LIN {X 0,Y 408.559,Z 372.352,A -85,B 0,C 180,E1 18045.699,E2 18045.699} C_VEL
LIN {X 0,Y 407.046,Z 362.331,A -85,B 0,C 180,E1 18045.227,E2 18045.227} C_VEL
LIN {X 0,Y 396.72,Z 344.882,A -85,B 0,C 180,E1 18043.129,E2 18043.129} C_VEL
LIN {X 0,Y 386.297,Z 328.726,A -85,B 0,C 180,E1 18040.835,E2 18040.835} C_VEL
LIN {X 0,Y 381.778,Z 321.934,A -85,B 0,C 180,E1 18039.72,E2 18039.72} C_VEL
LIN {X 0,Y 376.078,Z 309.997,A -85,B 0,C 180,E1 18036.741,E2 18036.741} C_VEL
LIN {X 0,Y 371.702,Z 301.451,A -85,B 0,C 180,E1 18034.331,E2 18034.331} C_VEL
LIN {X 0,Y 369.056,Z 296.536,A -85,B 0,C 180,E1 18032.81,E2 18032.81} C_VEL
LIN {X 0,Y 366.734,Z 292.115,A -85,B 0,C 180,E1 18031.382,E2 18031.382} C_VEL
LIN {X 0,Y 364.759,Z 288.388,A -85,B 0,C 180,E1 18030.108,E2 18030.108} C_VEL
LIN {X 0,Y 362.046,Z 283.882,A -85,B 0,C 180,E1 18028.36,E2 18028.36} C_VEL
LIN {X 0,Y 361.832,Z 282.774,A -85,B 0,C 180,E1 18027.84,E2 18027.84} C_VEL
LIN {X 0,Y 361.811,Z 282.657,A -85,B 0,C 180,E1 18023.623,E2 18023.623} C_VEL
LIN {X 0,Y 361.809,Z 282.653,A -85,B 0,C 180,E1 18019.535,E2 18019.535} C_VEL
LIN {X 0,Y 361.808,Z 282.65,A -85,B 0,C 180,E1 18015.327,E2 18015.327} C_VEL
LIN {X 0,Y 361.791,Z 282.651,A -85,B 0,C 180,E1 18011.155,E2 18011.155} C_VEL
LIN {X 0,Y 361.78,Z 282.655,A -85,B 0,C 180,E1 18006.985,E2 18006.985} C_VEL
LIN {X 0,Y 361.77,Z 282.662,A -85,B 0,C 180,E1 18002.852,E2 18002.852} C_VEL
LIN {X 0,Y 361.762,Z 282.669,A -85,B 0,C 180,E1 17998.733,E2 17998.733} C_VEL
LIN {X 0,Y 361.753,Z 282.674,A -85,B 0,C 180,E1 17994.608,E2 17994.608} C_VEL
LIN {X 0,Y 361.748,Z 282.675,A -85,B 0,C 180,E1 17990.615,E2 17990.615} C_VEL
LIN {X 0,Y 361.742,Z 282.675,A -85,B 0,C 180,E1 17986.575,E2 17986.575} C_VEL
LIN {X 0,Y 361.74,Z 282.674,A -85,B 0,C 180,E1 17982.466,E2 17982.466} C_VEL
LIN {X 0,Y 361.746,Z 282.671,A -85,B 0,C 180,E1 17978.432,E2 17978.432} C_VEL
LIN {X 0,Y 361.819,Z 282.907,A -85,B 0,C 180,E1 17975.163,E2 17975.163} C_VEL
LIN {X 0,Y 363.332,Z 286.523,A -85,B 0,C 180,E1 17973.877,E2 17973.877} C_VEL
LIN {X 0,Y 364.801,Z 288.276,A -85,B 0,C 180,E1 17973.113,E2 17973.113} C_VEL
LIN {X 0,Y 366.755,Z 292.174,A -85,B 0,C 180,E1 17971.86,E2 17971.86} C_VEL
LIN {X 0,Y 367.885,Z 293.939,A -85,B 0,C 180,E1 17971.246,E2 17971.246} C_VEL
LIN {X 0,Y 370.686,Z 299.01,A -85,B 0,C 180,E1 17969.668,E2 17969.668} C_VEL
LIN {X 0,Y 375.284,Z 307.456,A -85,B 0,C 180,E1 17967.259,E2 17967.259} C_VEL
LIN {X 0,Y 376.894,Z 310.291,A -85,B 0,C 180,E1 17966.646,E2 17966.646} C_VEL
LIN {X 0,Y 385.998,Z 322.591,A -85,B 0,C 180,E1 17964.442,E2 17964.442} C_VEL
LIN {X 0,Y 396.684,Z 338.125,A -85,B 0,C 180,E1 17962.073,E2 17962.073} C_VEL
LIN {X 0,Y 408.24,Z 356.697,A -85,B 0,C 180,E1 17959.716,E2 17959.716} C_VEL
LIN {X 0,Y 411.508,Z 362.693,A -85,B 0,C 180,E1 17959.072,E2 17959.072} C_VEL
LIN {X 0,Y 402.389,Z 573.786,A -85,B 0,C 180,E1 17954.935,E2 17954.935} C_VEL
LIN {X 0,Y 400.703,Z 607.918,A -85,B 0,C 180,E1 17954.213,E2 17954.213} C_VEL
LIN {X 0,Y 398.591,Z 630.344,A -85,B 0,C 180,E1 17953.522,E2 17953.522} C_VEL
LIN {X 0,Y 395.913,Z 651.73,A -85,B 0,C 180,E1 17952.594,E2 17952.594} C_VEL
LIN {X 0,Y 392.818,Z 672.423,A -85,B 0,C 180,E1 17951.435,E2 17951.435} C_VEL
LIN {X 0,Y 389.456,Z 691.906,A -85,B 0,C 180,E1 17950.088,E2 17950.088} C_VEL
LIN {X 0,Y 385.56,Z 711.788,A -85,B 0,C 180,E1 17948.394,E2 17948.394} C_VEL
LIN {X 0,Y 381.679,Z 730.327,A -85,B 0,C 180,E1 17946.487,E2 17946.487} C_VEL
LIN {X 0,Y 377.741,Z 748.111,A -85,B 0,C 180,E1 17944.318,E2 17944.318} C_VEL
LIN {X 0,Y 373.949,Z 765.002,A -85,B 0,C 180,E1 17941.874,E2 17941.874} C_VEL
LIN {X 0,Y 370.47,Z 780.284,A -85,B 0,C 180,E1 17939.241,E2 17939.241} C_VEL
LIN {X 0,Y 367.358,Z 794.572,A -85,B 0,C 180,E1 17936.336,E2 17936.336} C_VEL
LIN {X 0,Y 364.783,Z 807.38,A -85,B 0,C 180,E1 17933.246,E2 17933.246} C_VEL
LIN {X 0,Y 362.879,Z 818.173,A -85,B 0,C 180,E1 17930.146,E2 17930.146} C_VEL
LIN {X 0,Y 361.483,Z 827.462,A -85,B 0,C 180,E1 17926.883,E2 17926.883} C_VEL
LIN {X 0,Y 360.594,Z 835.304,A -85,B 0,C 180,E1 17923.468,E2 17923.468} C_VEL
LIN {X 0,Y 360.17,Z 841.103,A -85,B 0,C 180,E1 17920.234,E2 17920.234} C_VEL
LIN {X 0,Y 360.026,Z 845.162,A -85,B 0,C 180,E1 17917.019,E2 17917.019} C_VEL
LIN {X 0,Y 359.994,Z 847.849,A -85,B 0,C 180,E1 17913.662,E2 17913.662} C_VEL
LIN {X 0,Y 360.004,Z 848.78,A -85,B 0,C 180,E1 17910.796,E2 17910.796} C_VEL
LIN {X 0,Y 359.999,Z 848.431,A -85,B 0,C 180,E1 17907.612,E2 17907.612} C_VEL
LIN {X 0,Y 360.003,Z 846.641,A -85,B 0,C 180,E1 17904.582,E2 17904.582} C_VEL
LIN {X 0,Y 360.072,Z 843.093,A -85,B 0,C 180,E1 17901.215,E2 17901.215} C_VEL
LIN {X 0,Y 360.343,Z 838.399,A -85,B 0,C 180,E1 17898.151,E2 17898.151} C_VEL
LIN {X 0,Y 360.95,Z 831.803,A -85,B 0,C 180,E1 17894.907,E2 17894.907} C_VEL
LIN {X 0,Y 362.036,Z 823.526,A -85,B 0,C 180,E1 17891.649,E2 17891.649} C_VEL
LIN {X 0,Y 363.704,Z 813.284,A -85,B 0,C 180,E1 17888.385,E2 17888.385} C_VEL
LIN {X 0,Y 365.916,Z 801.567,A -85,B 0,C 180,E1 17885.288,E2 17885.288} C_VEL
LIN {X 0,Y 368.825,Z 787.697,A -85,B 0,C 180,E1 17882.208,E2 17882.208} C_VEL
LIN {X 0,Y 372.076,Z 773.156,A -85,B 0,C 180,E1 17879.478,E2 17879.478} C_VEL
LIN {X 0,Y 375.715,Z 757.109,A -85,B 0,C 180,E1 17876.939,E2 17876.939} C_VEL
LIN {X 0,Y 379.502,Z 740.143,A -85,B 0,C 180,E1 17874.67,E2 17874.67} C_VEL
LIN {X 0,Y 383.602,Z 721.198,A -85,B 0,C 180,E1 17872.537,E2 17872.537} C_VEL
LIN {X 0,Y 387.425,Z 702.563,A -85,B 0,C 180,E1 17870.782,E2 17870.782} C_VEL
LIN {X 0,Y 390.927,Z 683.359,A -85,B 0,C 180,E1 17869.293,E2 17869.293} C_VEL
LIN {X 0,Y 394.328,Z 662.52,A -85,B 0,C 180,E1 17867.981,E2 17867.981} C_VEL
LIN {X 0,Y 397.271,Z 641.356,A -85,B 0,C 180,E1 17866.929,E2 17866.929} C_VEL
LIN {X 0,Y 399.587,Z 620.581,A -85,B 0,C 180,E1 17866.155,E2 17866.155} C_VEL
LIN {X 0,Y 401.273,Z 598.399,A -85,B 0,C 180,E1 17865.57,E2 17865.57} C_VEL
LIN {X 0,Y 410.569,Z 383.446,A -85,B 0,C 180,E1 17861.338,E2 17861.338} C_VEL
LIN {X 0,Y 411.329,Z 362.088,A -85,B 0,C 180,E1 17860.897,E2 17860.897} C_VEL
LIN {X 0,Y 401.183,Z 345.219,A -85,B 0,C 180,E1 17858.883,E2 17858.883} C_VEL
LIN {X 0,Y 390.845,Z 329.535,A -85,B 0,C 180,E1 17856.679,E2 17856.679} C_VEL
LIN {X 0,Y 381.262,Z 316.025,A -85,B 0,C 180,E1 17854.458,E2 17854.458} C_VEL
LIN {X 0,Y 375.815,Z 308.655,A -85,B 0,C 180,E1 17853.052,E2 17853.052} C_VEL
LIN {X 0,Y 372.269,Z 301.954,A -85,B 0,C 180,E1 17851.223,E2 17851.223} C_VEL
LIN {X 0,Y 369.727,Z 297.293,A -85,B 0,C 180,E1 17849.841,E2 17849.841} C_VEL
LIN {X 0,Y 366.999,Z 292.443,A -85,B 0,C 180,E1 17848.297,E2 17848.297} C_VEL
LIN {X 0,Y 364.933,Z 288.721,A -85,B 0,C 180,E1 17847.053,E2 17847.053} C_VEL
LIN {X 0,Y 363.842,Z 287.108,A -85,B 0,C 180,E1 17846.435,E2 17846.435} C_VEL
LIN {X 0,Y 362.104,Z 284.18,A -85,B 0,C 180,E1 17845.34,E2 17845.34} C_VEL
LIN {X 0,Y 361.813,Z 282.858,A -85,B 0,C 180,E1 17844.837,E2 17844.837} C_VEL
LIN {X 0,Y 361.785,Z 282.663,A -85,B 0,C 180,E1 17840.886,E2 17840.886} C_VEL
LIN {X 0,Y 361.775,Z 282.657,A -85,B 0,C 180,E1 17836.704,E2 17836.704} C_VEL
LIN {X 0,Y 361.771,Z 282.657,A -85,B 0,C 180,E1 17832.611,E2 17832.611} C_VEL
LIN {X 0,Y 361.769,Z 282.659,A -85,B 0,C 180,E1 17828.423,E2 17828.423} C_VEL
LIN {X 0,Y 361.776,Z 282.665,A -85,B 0,C 180,E1 17824.438,E2 17824.438} C_VEL
LIN {X 0,Y 361.777,Z 282.669,A -85,B 0,C 180,E1 17820.316,E2 17820.316} C_VEL
LIN {X 0,Y 361.777,Z 282.672,A -85,B 0,C 180,E1 17816.196,E2 17816.196} C_VEL
LIN {X 0,Y 361.778,Z 282.672,A -85,B 0,C 180,E1 17812.057,E2 17812.057} C_VEL
LIN {X 0,Y 361.774,Z 282.671,A -85,B 0,C 180,E1 17807.875,E2 17807.875} C_VEL
LIN {X 0,Y 361.779,Z 282.668,A -85,B 0,C 180,E1 17803.791,E2 17803.791} C_VEL
LIN {X 0,Y 361.781,Z 282.67,A -85,B 0,C 180,E1 17799.621,E2 17799.621} C_VEL
LIN {X 0,Y 361.784,Z 282.669,A -85,B 0,C 180,E1 17795.399,E2 17795.399} C_VEL
LIN {X 0,Y 361.829,Z 282.875,A -85,B 0,C 180,E1 17791.875,E2 17791.875} C_VEL
LIN {X 0,Y 363.175,Z 286.201,A -85,B 0,C 180,E1 17790.656,E2 17790.656} C_VEL
LIN {X 0,Y 364.832,Z 288.623,A -85,B 0,C 180,E1 17789.685,E2 17789.685} C_VEL
LIN {X 0,Y 366.815,Z 292.212,A -85,B 0,C 180,E1 17788.442,E2 17788.442} C_VEL
LIN {X 0,Y 370.235,Z 298.661,A -85,B 0,C 180,E1 17786.384,E2 17786.384} C_VEL
LIN {X 0,Y 374.748,Z 307.279,A -85,B 0,C 180,E1 17783.868,E2 17783.868} C_VEL
LIN {X 0,Y 380.66,Z 319.547,A -85,B 0,C 180,E1 17780.726,E2 17780.726} C_VEL
LIN {X 0,Y 382.582,Z 323.315,A -85,B 0,C 180,E1 17779.917,E2 17779.917} C_VEL
LIN {X 0,Y 394.621,Z 341.47,A -85,B 0,C 180,E1 17777.206,E2 17777.206} C_VEL
LIN {X 0,Y 405.534,Z 359.797,A -85,B 0,C 180,E1 17774.959,E2 17774.959} C_VEL
LIN {X 0,Y 407.24,Z 363.206,A -85,B 0,C 180,E1 17774.613,E2 17774.613} C_VEL
LIN {X 0,Y 408.507,Z 373.825,A -85,B 0,C 180,E1 17774.166,E2 17774.166} C_VEL
LIN {X 0,Y 400.581,Z 595.446,A -85,B 0,C 180,E1 17770.128,E2 17770.128} C_VEL
LIN {X 0,Y 398.92,Z 616.173,A -85,B 0,C 180,E1 17769.518,E2 17769.518} C_VEL
LIN {X 0,Y 396.654,Z 635.991,A -85,B 0,C 180,E1 17768.691,E2 17768.691} C_VEL
LIN {X 0,Y 393.787,Z 655.659,A -85,B 0,C 180,E1 17767.608,E2 17767.608} C_VEL
LIN {X 0,Y 390.647,Z 673.719,A -85,B 0,C 180,E1 17766.354,E2 17766.354} C_VEL
LIN {X 0,Y 387.043,Z 691.567,A -85,B 0,C 180,E1 17764.813,E2 17764.813} C_VEL
LIN {X 0,Y 383.227,Z 708.408,A -85,B 0,C 180,E1 17763.044,E2 17763.044} C_VEL
LIN {X 0,Y 379.18,Z 724.954,A -85,B 0,C 180,E1 17760.943,E2 17760.943} C_VEL
LIN {X 0,Y 375.312,Z 739.918,A -85,B 0,C 180,E1 17758.654,E2 17758.654} C_VEL
LIN {X 0,Y 371.752,Z 753.448,A -85,B 0,C 180,E1 17756.173,E2 17756.173} C_VEL
LIN {X 0,Y 368.381,Z 766.177,A -85,B 0,C 180,E1 17753.345,E2 17753.345} C_VEL
LIN {X 0,Y 365.69,Z 776.731,A -85,B 0,C 180,E1 17750.485,E2 17750.485} C_VEL
LIN {X 0,Y 363.471,Z 786.215,A -85,B 0,C 180,E1 17747.34,E2 17747.34} C_VEL
LIN {X 0,Y 361.885,Z 794.048,A -85,B 0,C 180,E1 17744.071,E2 17744.071} C_VEL
LIN {X 0,Y 361.143,Z 798.41,A -85,B 0,C 180,E1 17741.796,E2 17741.796} C_VEL
LIN {X 0,Y 359.88,Z 800.467,A -85,B 0,C 180,E1 17740.624,E2 17740.624} C_VEL
LIN {X 0,Y 353.022,Z 805.15,A -85,B 0,C 180,E1 17737.373,E2 17737.373} C_VEL
LIN {X 0,Y 352.29,Z 806.085,A -85,B 0,C 180,E1 17736.396,E2 17736.396} C_VEL
LIN {X 0,Y 352.114,Z 808.279,A -85,B 0,C 180,E1 17732.93,E2 17732.93} C_VEL
LIN {X 0,Y 352.084,Z 808.901,A -85,B 0,C 180,E1 17729.675,E2 17729.675} C_VEL
LIN {X 0,Y 352.129,Z 808.066,A -85,B 0,C 180,E1 17726.419,E2 17726.419} C_VEL
LIN {X 0,Y 352.319,Z 805.768,A -85,B 0,C 180,E1 17723.155,E2 17723.155} C_VEL
LIN {X 0,Y 352.805,Z 801.779,A -85,B 0,C 180,E1 17719.715,E2 17719.715} C_VEL
LIN {X 0,Y 353.7,Z 796.383,A -85,B 0,C 180,E1 17716.431,E2 17716.431} C_VEL
LIN {X 0,Y 355.283,Z 788.833,A -85,B 0,C 180,E1 17712.982,E2 17712.982} C_VEL
LIN {X 0,Y 357.501,Z 779.638,A -85,B 0,C 180,E1 17709.709,E2 17709.709} C_VEL
LIN {X 0,Y 360.209,Z 769.371,A -85,B 0,C 180,E1 17706.749,E2 17706.749} C_VEL
LIN {X 0,Y 363.542,Z 757.357,A -85,B 0,C 180,E1 17703.894,E2 17703.894} C_VEL
LIN {X 0,Y 367.143,Z 744.548,A -85,B 0,C 180,E1 17701.361,E2 17701.361} C_VEL
LIN {X 0,Y 371.241,Z 729.73,A -85,B 0,C 180,E1 17698.922,E2 17698.922} C_VEL
LIN {X 0,Y 375.443,Z 713.556,A -85,B 0,C 180,E1 17696.73,E2 17696.73} C_VEL
LIN {X 0,Y 379.489,Z 696.764,A -85,B 0,C 180,E1 17694.853,E2 17694.853} C_VEL
LIN {X 0,Y 383.437,Z 678.576,A -85,B 0,C 180,E1 17693.182,E2 17693.182} C_VEL
LIN {X 0,Y 386.84,Z 660.766,A -85,B 0,C 180,E1 17691.85,E2 17691.85} C_VEL
LIN {X 0,Y 389.931,Z 641.542,A -85,B 0,C 180,E1 17690.703,E2 17690.703} C_VEL
LIN {X 0,Y 392.484,Z 621.377,A -85,B 0,C 180,E1 17689.796,E2 17689.796} C_VEL
LIN {X 0,Y 394.345,Z 600.962,A -85,B 0,C 180,E1 17689.134,E2 17689.134} C_VEL
LIN {X 0,Y 395.679,Z 573.766,A -85,B 0,C 180,E1 17688.565,E2 17688.565} C_VEL
LIN {X 0,Y 403.042,Z 373.798,A -85,B 0,C 180,E1 17684.893,E2 17684.893} C_VEL
LIN {X 0,Y 401.891,Z 366.492,A -85,B 0,C 180,E1 17684.53,E2 17684.53} C_VEL
LIN {X 0,Y 392.227,Z 349.993,A -85,B 0,C 180,E1 17682.496,E2 17682.496} C_VEL
LIN {X 0,Y 382.017,Z 333.999,A -85,B 0,C 180,E1 17680.169,E2 17680.169} C_VEL
LIN {X 0,Y 373.505,Z 321.545,A -85,B 0,C 180,E1 17678.003,E2 17678.003} C_VEL
LIN {X 0,Y 368.505,Z 311.291,A -85,B 0,C 180,E1 17675.247,E2 17675.247} C_VEL
LIN {X 0,Y 364.257,Z 302.957,A -85,B 0,C 180,E1 17672.735,E2 17672.735} C_VEL
LIN {X 0,Y 361.662,Z 298.135,A -85,B 0,C 180,E1 17671.131,E2 17671.131} C_VEL
LIN {X 0,Y 359.22,Z 293.573,A -85,B 0,C 180,E1 17669.516,E2 17669.516} C_VEL
LIN {X 0,Y 357.062,Z 289.858,A -85,B 0,C 180,E1 17668.063,E2 17668.063} C_VEL
LIN {X 0,Y 356.124,Z 288.304,A -85,B 0,C 180,E1 17667.416,E2 17667.416} C_VEL
LIN {X 0,Y 354.132,Z 284.926,A -85,B 0,C 180,E1 17665.953,E2 17665.953} C_VEL
LIN {X 0,Y 353.888,Z 283.8,A -85,B 0,C 180,E1 17665.433,E2 17665.433} C_VEL
LIN {X 0,Y 353.87,Z 283.643,A -85,B 0,C 180,E1 17661.376,E2 17661.376} C_VEL
LIN {X 0,Y 353.862,Z 283.647,A -85,B 0,C 180,E1 17657.251,E2 17657.251} C_VEL
LIN {X 0,Y 353.851,Z 283.648,A -85,B 0,C 180,E1 17653.065,E2 17653.065} C_VEL
LIN {X 0,Y 353.84,Z 283.646,A -85,B 0,C 180,E1 17648.941,E2 17648.941} C_VEL
LIN {X 0,Y 353.832,Z 283.643,A -85,B 0,C 180,E1 17644.863,E2 17644.863} C_VEL
LIN {X 0,Y 353.826,Z 283.64,A -85,B 0,C 180,E1 17640.81,E2 17640.81} C_VEL
LIN {X 0,Y 353.82,Z 283.639,A -85,B 0,C 180,E1 17636.76,E2 17636.76} C_VEL
LIN {X 0,Y 353.813,Z 283.639,A -85,B 0,C 180,E1 17632.694,E2 17632.694} C_VEL
LIN {X 0,Y 353.804,Z 283.64,A -85,B 0,C 180,E1 17628.591,E2 17628.591} C_VEL
LIN {X 0,Y 353.794,Z 283.641,A -85,B 0,C 180,E1 17624.426,E2 17624.426} C_VEL
LIN {X 0,Y 353.799,Z 283.643,A -85,B 0,C 180,E1 17620.177,E2 17620.177} C_VEL
LIN {X 0,Y 353.876,Z 284.009,A -85,B 0,C 180,E1 17617.578,E2 17617.578} C_VEL
LIN {X 0,Y 355.542,Z 287.711,A -85,B 0,C 180,E1 17616.112,E2 17616.112} C_VEL
LIN {X 0,Y 356.945,Z 289.23,A -85,B 0,C 180,E1 17615.332,E2 17615.332} C_VEL
LIN {X 0,Y 358.676,Z 292.941,A -85,B 0,C 180,E1 17614.046,E2 17614.046} C_VEL
LIN {X 0,Y 360.054,Z 294.855,A -85,B 0,C 180,E1 17613.265,E2 17613.265} C_VEL
LIN {X 0,Y 362.059,Z 298.589,A -85,B 0,C 180,E1 17612,E2 17612} C_VEL
LIN {X 0,Y 363.339,Z 301.047,A -85,B 0,C 180,E1 17611.212,E2 17611.212} C_VEL
LIN {X 0,Y 365.828,Z 305.453,A -85,B 0,C 180,E1 17609.808,E2 17609.808} C_VEL
LIN {X 0,Y 368.266,Z 309.707,A -85,B 0,C 180,E1 17608.582,E2 17608.582} C_VEL
LIN {X 0,Y 379.261,Z 324.47,A -85,B 0,C 180,E1 17605.701,E2 17605.701} C_VEL
LIN {X 0,Y 389.526,Z 339.289,A -85,B 0,C 180,E1 17603.291,E2 17603.291} C_VEL
LIN {X 0,Y 400.953,Z 357.285,A -85,B 0,C 180,E1 17600.837,E2 17600.837} C_VEL
LIN {X 0,Y 405.886,Z 366.065,A -85,B 0,C 180,E1 17599.828,E2 17599.828} C_VEL
LIN {X 0,Y 396.319,Z 578.508,A -85,B 0,C 180,E1 17595.625,E2 17595.625} C_VEL
LIN {X 0,Y 394.662,Z 609.067,A -85,B 0,C 180,E1 17594.957,E2 17594.957} C_VEL
LIN {X 0,Y 392.467,Z 631.269,A -85,B 0,C 180,E1 17594.256,E2 17594.256} C_VEL
LIN {X 0,Y 389.727,Z 652.133,A -85,B 0,C 180,E1 17593.335,E2 17593.335} C_VEL
LIN {X 0,Y 386.508,Z 672.676,A -85,B 0,C 180,E1 17592.166,E2 17592.166} C_VEL
LIN {X 0,Y 382.961,Z 692.287,A -85,B 0,C 180,E1 17590.787,E2 17590.787} C_VEL
LIN {X 0,Y 378.949,Z 711.885,A -85,B 0,C 180,E1 17589.093,E2 17589.093} C_VEL
LIN {X 0,Y 374.886,Z 730.347,A -85,B 0,C 180,E1 17587.163,E2 17587.163} C_VEL
LIN {X 0,Y 370.623,Z 748.64,A -85,B 0,C 180,E1 17584.884,E2 17584.884} C_VEL
LIN {X 0,Y 366.771,Z 764.903,A -85,B 0,C 180,E1 17582.482,E2 17582.482} C_VEL
LIN {X 0,Y 363.011,Z 780.59,A -85,B 0,C 180,E1 17579.72,E2 17579.72} C_VEL
LIN {X 0,Y 359.875,Z 794.16,A -85,B 0,C 180,E1 17576.894,E2 17576.894} C_VEL
LIN {X 0,Y 357.157,Z 806.852,A -85,B 0,C 180,E1 17573.773,E2 17573.773} C_VEL
LIN {X 0,Y 355.116,Z 817.654,A -85,B 0,C 180,E1 17570.606,E2 17570.606} C_VEL
LIN {X 0,Y 353.616,Z 826.961,A -85,B 0,C 180,E1 17567.27,E2 17567.27} C_VEL
LIN {X 0,Y 352.651,Z 834.82,A -85,B 0,C 180,E1 17563.778,E2 17563.778} C_VEL
LIN {X 0,Y 352.194,Z 840.631,A -85,B 0,C 180,E1 17560.468,E2 17560.468} C_VEL
LIN {X 0,Y 352.034,Z 844.702,A -85,B 0,C 180,E1 17557.179,E2 17557.179} C_VEL
LIN {X 0,Y 352.001,Z 847.324,A -85,B 0,C 180,E1 17553.909,E2 17553.909} C_VEL
LIN {X 0,Y 352.017,Z 848.332,A -85,B 0,C 180,E1 17550.814,E2 17550.814} C_VEL
LIN {X 0,Y 352.009,Z 847.981,A -85,B 0,C 180,E1 17547.558,E2 17547.558} C_VEL
LIN {X 0,Y 352.008,Z 846.186,A -85,B 0,C 180,E1 17544.458,E2 17544.458} C_VEL
LIN {X 0,Y 352.085,Z 842.625,A -85,B 0,C 180,E1 17541.014,E2 17541.014} C_VEL
LIN {X 0,Y 352.379,Z 837.922,A -85,B 0,C 180,E1 17537.88,E2 17537.88} C_VEL
LIN {X 0,Y 353.039,Z 831.309,A -85,B 0,C 180,E1 17534.561,E2 17534.561} C_VEL
LIN {X 0,Y 354.209,Z 823.014,A -85,B 0,C 180,E1 17531.229,E2 17531.229} C_VEL
LIN {X 0,Y 355.952,Z 812.998,A -85,B 0,C 180,E1 17527.965,E2 17527.965} C_VEL
LIN {X 0,Y 358.224,Z 801.692,A -85,B 0,C 180,E1 17524.897,E2 17524.897} C_VEL
LIN {X 0,Y 361.105,Z 788.74,A -85,B 0,C 180,E1 17521.92,E2 17521.92} C_VEL
LIN {X 0,Y 364.476,Z 774.408,A -85,B 0,C 180,E1 17519.138,E2 17519.138} C_VEL
LIN {X 0,Y 368.242,Z 758.602,A -85,B 0,C 180,E1 17516.552,E2 17516.552} C_VEL
LIN {X 0,Y 372.459,Z 740.748,A -85,B 0,C 180,E1 17514.088,E2 17514.088} C_VEL
LIN {X 0,Y 376.622,Z 722.553,A -85,B 0,C 180,E1 17511.983,E2 17511.983} C_VEL
LIN {X 0,Y 380.711,Z 703.522,A -85,B 0,C 180,E1 17510.149,E2 17510.149} C_VEL
LIN {X 0,Y 384.54,Z 683.543,A -85,B 0,C 180,E1 17508.569,E2 17508.569} C_VEL
LIN {X 0,Y 388.184,Z 662.187,A -85,B 0,C 180,E1 17507.209,E2 17507.209} C_VEL
LIN {X 0,Y 391.234,Z 641.045,A -85,B 0,C 180,E1 17506.152,E2 17506.152} C_VEL
LIN {X 0,Y 393.62,Z 620.423,A -85,B 0,C 180,E1 17505.379,E2 17505.379} C_VEL
LIN {X 0,Y 395.364,Z 598.238,A -85,B 0,C 180,E1 17504.789,E2 17504.789} C_VEL
LIN {X 0,Y 405.037,Z 383.817,A -85,B 0,C 180,E1 17500.527,E2 17500.527} C_VEL
LIN {X 0,Y 405.745,Z 365.58,A -85,B 0,C 180,E1 17500.151,E2 17500.151} C_VEL
LIN {X 0,Y 395.168,Z 347.98,A -85,B 0,C 180,E1 17497.963,E2 17497.963} C_VEL
LIN {X 0,Y 384.1,Z 331.343,A -85,B 0,C 180,E1 17495.485,E2 17495.485} C_VEL
LIN {X 0,Y 374.395,Z 317.884,A -85,B 0,C 180,E1 17493.102,E2 17493.102} C_VEL
LIN {X 0,Y 367.851,Z 308.914,A -85,B 0,C 180,E1 17491.275,E2 17491.275} C_VEL
LIN {X 0,Y 364.372,Z 302.868,A -85,B 0,C 180,E1 17489.418,E2 17489.418} C_VEL
LIN {X 0,Y 362.299,Z 298.857,A -85,B 0,C 180,E1 17488.159,E2 17488.159} C_VEL
LIN {X 0,Y 360.193,Z 295.27,A -85,B 0,C 180,E1 17486.902,E2 17486.902} C_VEL
LIN {X 0,Y 359.177,Z 293.529,A -85,B 0,C 180,E1 17486.271,E2 17486.271} C_VEL
LIN {X 0,Y 357.226,Z 290.153,A -85,B 0,C 180,E1 17485.001,E2 17485.001} C_VEL
LIN {X 0,Y 356.582,Z 288.805,A -85,B 0,C 180,E1 17484.519,E2 17484.519} C_VEL
LIN {X 0,Y 354.351,Z 285.638,A -85,B 0,C 180,E1 17483.092,E2 17483.092} C_VEL
LIN {X 0,Y 353.845,Z 283.832,A -85,B 0,C 180,E1 17482.331,E2 17482.331} C_VEL
LIN {X 0,Y 353.814,Z 283.649,A -85,B 0,C 180,E1 17478.281,E2 17478.281} C_VEL
LIN {X 0,Y 353.807,Z 283.651,A -85,B 0,C 180,E1 17474.232,E2 17474.232} C_VEL
LIN {X 0,Y 353.807,Z 283.653,A -85,B 0,C 180,E1 17470.091,E2 17470.091} C_VEL
LIN {X 0,Y 353.811,Z 283.65,A -85,B 0,C 180,E1 17466.002,E2 17466.002} C_VEL
LIN {X 0,Y 353.813,Z 283.645,A -85,B 0,C 180,E1 17461.943,E2 17461.943} C_VEL
LIN {X 0,Y 353.819,Z 283.64,A -85,B 0,C 180,E1 17457.894,E2 17457.894} C_VEL
LIN {X 0,Y 353.823,Z 283.637,A -85,B 0,C 180,E1 17453.835,E2 17453.835} C_VEL
LIN {X 0,Y 353.827,Z 283.637,A -85,B 0,C 180,E1 17449.745,E2 17449.745} C_VEL
LIN {X 0,Y 353.829,Z 283.638,A -85,B 0,C 180,E1 17445.601,E2 17445.601} C_VEL
LIN {X 0,Y 353.836,Z 283.638,A -85,B 0,C 180,E1 17441.378,E2 17441.378} C_VEL
LIN {X 0,Y 353.843,Z 283.639,A -85,B 0,C 180,E1 17437.224,E2 17437.224} C_VEL
LIN {X 0,Y 353.911,Z 283.942,A -85,B 0,C 180,E1 17434.266,E2 17434.266} C_VEL
LIN {X 0,Y 355.366,Z 287.416,A -85,B 0,C 180,E1 17432.883,E2 17432.883} C_VEL
LIN {X 0,Y 356.92,Z 289.439,A -85,B 0,C 180,E1 17431.925,E2 17431.925} C_VEL
LIN {X 0,Y 358.709,Z 292.962,A -85,B 0,C 180,E1 17430.621,E2 17430.621} C_VEL
LIN {X 0,Y 359.771,Z 294.532,A -85,B 0,C 180,E1 17429.983,E2 17429.983} C_VEL
LIN {X 0,Y 362.043,Z 298.611,A -85,B 0,C 180,E1 17428.536,E2 17428.536} C_VEL
LIN {X 0,Y 365.607,Z 305.796,A -85,B 0,C 180,E1 17426.278,E2 17426.278} C_VEL
LIN {X 0,Y 369.295,Z 312.696,A -85,B 0,C 180,E1 17424.21,E2 17424.21} C_VEL
LIN {X 0,Y 373.949,Z 322.392,A -85,B 0,C 180,E1 17421.709,E2 17421.709} C_VEL
LIN {X 0,Y 383.134,Z 335.742,A -85,B 0,C 180,E1 17419.448,E2 17419.448} C_VEL
LIN {X 0,Y 394.167,Z 353.169,A -85,B 0,C 180,E1 17416.972,E2 17416.972} C_VEL
LIN {X 0,Y 402.093,Z 367.173,A -85,B 0,C 180,E1 17415.311,E2 17415.311} C_VEL
LIN {X 0,Y 402.99,Z 375.353,A -85,B 0,C 180,E1 17414.968,E2 17414.968} C_VEL
LIN {X 0,Y 394.7,Z 595.554,A -85,B 0,C 180,E1 17410.912,E2 17410.912} C_VEL
LIN {X 0,Y 392.966,Z 616.343,A -85,B 0,C 180,E1 17410.295,E2 17410.295} C_VEL
LIN {X 0,Y 390.592,Z 636.311,A -85,B 0,C 180,E1 17409.455,E2 17409.455} C_VEL
LIN {X 0,Y 387.573,Z 656.181,A -85,B 0,C 180,E1 17408.348,E2 17408.348} C_VEL
LIN {X 0,Y 384.155,Z 674.898,A -85,B 0,C 180,E1 17407.023,E2 17407.023} C_VEL
LIN {X 0,Y 380.297,Z 693.237,A -85,B 0,C 180,E1 17405.408,E2 17405.408} C_VEL
LIN {X 0,Y 376.21,Z 710.335,A -85,B 0,C 180,E1 17403.559,E2 17403.559} C_VEL
LIN {X 0,Y 372.153,Z 726.071,A -85,B 0,C 180,E1 17401.503,E2 17401.503} C_VEL
LIN {X 0,Y 367.993,Z 741.356,A -85,B 0,C 180,E1 17399.1,E2 17399.1} C_VEL
LIN {X 0,Y 364.287,Z 754.708,A -85,B 0,C 180,E1 17396.575,E2 17396.575} C_VEL
LIN {X 0,Y 360.954,Z 766.688,A -85,B 0,C 180,E1 17393.854,E2 17393.854} C_VEL
LIN {X 0,Y 357.97,Z 777.772,A -85,B 0,C 180,E1 17390.776,E2 17390.776} C_VEL
LIN {X 0,Y 355.698,Z 786.905,A -85,B 0,C 180,E1 17387.65,E2 17387.65} C_VEL
LIN {X 0,Y 354.047,Z 794.534,A -85,B 0,C 180,E1 17384.381,E2 17384.381} C_VEL
LIN {X 0,Y 353.003,Z 800.445,A -85,B 0,C 180,E1 17381.105,E2 17381.105} C_VEL
LIN {X 0,Y 352.413,Z 804.925,A -85,B 0,C 180,E1 17377.663,E2 17377.663} C_VEL
LIN {X 0,Y 352.29,Z 806.085,A -85,B 0,C 180,E1 17376.396,E2 17376.396} C_VEL
LIN {X 0,Y 351.212,Z 807.163,A -85,B 0,C 180,E1 17375.157,E2 17375.157} C_VEL
LIN {X 0,Y 346.508,Z 808.694,A -85,B 0,C 180,E1 17372.807,E2 17372.807} C_VEL
LIN {X 0,Y 344.311,Z 809.208,A -85,B 0,C 180,E1 17371.271,E2 17371.271} C_VEL
LIN {X 0,Y 344.099,Z 809.287,A -85,B 0,C 180,E1 17370.713,E2 17370.713} C_VEL
LIN {X 0,Y 344.118,Z 808.893,A -85,B 0,C 180,E1 17367.335,E2 17367.335} C_VEL
LIN {X 0,Y 344.268,Z 807.114,A -85,B 0,C 180,E1 17363.999,E2 17363.999} C_VEL
LIN {X 0,Y 344.693,Z 803.569,A -85,B 0,C 180,E1 17360.483,E2 17360.483} C_VEL
LIN {X 0,Y 345.497,Z 798.603,A -85,B 0,C 180,E1 17357.125,E2 17357.125} C_VEL
LIN {X 0,Y 346.977,Z 791.608,A -85,B 0,C 180,E1 17353.597,E2 17353.597} C_VEL
LIN {X 0,Y 348.986,Z 783.554,A -85,B 0,C 180,E1 17350.415,E2 17350.415} C_VEL
LIN {X 0,Y 351.721,Z 773.638,A -85,B 0,C 180,E1 17347.257,E2 17347.257} C_VEL
LIN {X 0,Y 355.029,Z 762.187,A -85,B 0,C 180,E1 17344.298,E2 17344.298} C_VEL
LIN {X 0,Y 358.58,Z 750.101,A -85,B 0,C 180,E1 17341.705,E2 17341.705} C_VEL
LIN {X 0,Y 362.73,Z 735.877,A -85,B 0,C 180,E1 17339.157,E2 17339.157} C_VEL
LIN {X 0,Y 366.94,Z 720.942,A -85,B 0,C 180,E1 17336.929,E2 17336.929} C_VEL
LIN {X 0,Y 371.24,Z 704.488,A -85,B 0,C 180,E1 17334.9,E2 17334.9} C_VEL
LIN {X 0,Y 375.291,Z 687.431,A -85,B 0,C 180,E1 17333.171,E2 17333.171} C_VEL
LIN {X 0,Y 379.242,Z 668.712,A -85,B 0,C 180,E1 17331.62,E2 17331.62} C_VEL
LIN {X 0,Y 382.601,Z 650.128,A -85,B 0,C 180,E1 17330.385,E2 17330.385} C_VEL
LIN {X 0,Y 385.461,Z 630.808,A -85,B 0,C 180,E1 17329.379,E2 17329.379} C_VEL
LIN {X 0,Y 387.747,Z 610.25,A -85,B 0,C 180,E1 17328.593,E2 17328.593} C_VEL
LIN {X 0,Y 389.27,Z 589.458,A -85,B 0,C 180,E1 17328.053,E2 17328.053} C_VEL
LIN {X 0,Y 397.612,Z 375.314,A -85,B 0,C 180,E1 17324.068,E2 17324.068} C_VEL
LIN {X 0,Y 396.873,Z 370.73,A -85,B 0,C 180,E1 17323.829,E2 17323.829} C_VEL
LIN {X 0,Y 386.274,Z 352.543,A -85,B 0,C 180,E1 17321.502,E2 17321.502} C_VEL
LIN {X 0,Y 374.631,Z 334.583,A -85,B 0,C 180,E1 17318.697,E2 17318.697} C_VEL
LIN {X 0,Y 365.305,Z 321.234,A -85,B 0,C 180,E1 17316.157,E2 17316.157} C_VEL
LIN {X 0,Y 360.964,Z 312.651,A -85,B 0,C 180,E1 17313.642,E2 17313.642} C_VEL
LIN {X 0,Y 358.595,Z 308.076,A -85,B 0,C 180,E1 17312.179,E2 17312.179} C_VEL
LIN {X 0,Y 356.609,Z 304.154,A -85,B 0,C 180,E1 17310.871,E2 17310.871} C_VEL
LIN {X 0,Y 354.192,Z 299.634,A -85,B 0,C 180,E1 17309.234,E2 17309.234} C_VEL
LIN {X 0,Y 352.116,Z 295.853,A -85,B 0,C 180,E1 17307.755,E2 17307.755} C_VEL
LIN {X 0,Y 349.399,Z 291.373,A -85,B 0,C 180,E1 17305.784,E2 17305.784} C_VEL
LIN {X 0,Y 348.648,Z 289.764,A -85,B 0,C 180,E1 17305.115,E2 17305.115} C_VEL
LIN {X 0,Y 346.386,Z 286.466,A -85,B 0,C 180,E1 17303.38,E2 17303.38} C_VEL
LIN {X 0,Y 345.937,Z 284.858,A -85,B 0,C 180,E1 17302.607,E2 17302.607} C_VEL
LIN {X 0,Y 345.9,Z 284.626,A -85,B 0,C 180,E1 17298.54,E2 17298.54} C_VEL
LIN {X 0,Y 345.895,Z 284.626,A -85,B 0,C 180,E1 17294.395,E2 17294.395} C_VEL
LIN {X 0,Y 345.895,Z 284.624,A -85,B 0,C 180,E1 17290.156,E2 17290.156} C_VEL
LIN {X 0,Y 345.89,Z 284.625,A -85,B 0,C 180,E1 17286.085,E2 17286.085} C_VEL
LIN {X 0,Y 345.887,Z 284.627,A -85,B 0,C 180,E1 17281.988,E2 17281.988} C_VEL
LIN {X 0,Y 345.886,Z 284.63,A -85,B 0,C 180,E1 17277.847,E2 17277.847} C_VEL
LIN {X 0,Y 345.89,Z 284.632,A -85,B 0,C 180,E1 17273.694,E2 17273.694} C_VEL
LIN {X 0,Y 345.889,Z 284.632,A -85,B 0,C 180,E1 17269.507,E2 17269.507} C_VEL
LIN {X 0,Y 345.906,Z 284.627,A -85,B 0,C 180,E1 17265.264,E2 17265.264} C_VEL
LIN {X 0,Y 345.896,Z 284.707,A -85,B 0,C 180,E1 17260.935,E2 17260.935} C_VEL
LIN {X 0,Y 345.935,Z 285.098,A -85,B 0,C 180,E1 17260.411,E2 17260.411} C_VEL
LIN {X 0,Y 347.714,Z 288.834,A -85,B 0,C 180,E1 17258.692,E2 17258.692} C_VEL
LIN {X 0,Y 349.299,Z 290.841,A -85,B 0,C 180,E1 17257.623,E2 17257.623} C_VEL
LIN {X 0,Y 351.186,Z 294.447,A -85,B 0,C 180,E1 17256.154,E2 17256.154} C_VEL
LIN {X 0,Y 352.248,Z 295.759,A -85,B 0,C 180,E1 17255.517,E2 17255.517} C_VEL
LIN {X 0,Y 354.29,Z 299.699,A -85,B 0,C 180,E1 17254.06,E2 17254.06} C_VEL
LIN {X 0,Y 355.311,Z 301.382,A -85,B 0,C 180,E1 17253.421,E2 17253.421} C_VEL
LIN {X 0,Y 358.113,Z 306.475,A -85,B 0,C 180,E1 17251.664,E2 17251.664} C_VEL
LIN {X 0,Y 360.64,Z 310.585,A -85,B 0,C 180,E1 17250.384,E2 17250.384} C_VEL
LIN {X 0,Y 369.303,Z 321.967,A -85,B 0,C 180,E1 17247.905,E2 17247.905} C_VEL
LIN {X 0,Y 378.881,Z 335.321,A -85,B 0,C 180,E1 17245.433,E2 17245.433} C_VEL
LIN {X 0,Y 388.953,Z 350.405,A -85,B 0,C 180,E1 17243.067,E2 17243.067} C_VEL
LIN {X 0,Y 399.715,Z 368.181,A -85,B 0,C 180,E1 17240.739,E2 17240.739} C_VEL
LIN {X 0,Y 400.322,Z 369.737,A -85,B 0,C 180,E1 17240.6,E2 17240.6} C_VEL
LIN {X 0,Y 390.238,Z 584.904,A -85,B 0,C 180,E1 17236.302,E2 17236.302} C_VEL
LIN {X 0,Y 388.587,Z 611.35,A -85,B 0,C 180,E1 17235.693,E2 17235.693} C_VEL
LIN {X 0,Y 386.233,Z 633.415,A -85,B 0,C 180,E1 17234.961,E2 17234.961} C_VEL
LIN {X 0,Y 383.342,Z 654.498,A -85,B 0,C 180,E1 17234.002,E2 17234.002} C_VEL
LIN {X 0,Y 380.006,Z 674.401,A -85,B 0,C 180,E1 17232.826,E2 17232.826} C_VEL
LIN {X 0,Y 376.099,Z 694.663,A -85,B 0,C 180,E1 17231.347,E2 17231.347} C_VEL
LIN {X 0,Y 371.958,Z 714.014,A -85,B 0,C 180,E1 17229.623,E2 17229.623} C_VEL
LIN {X 0,Y 367.672,Z 732.437,A -85,B 0,C 180,E1 17227.625,E2 17227.625} C_VEL
LIN {X 0,Y 363.398,Z 749.749,A -85,B 0,C 180,E1 17225.391,E2 17225.391} C_VEL
LIN {X 0,Y 359.26,Z 766.249,A -85,B 0,C 180,E1 17222.867,E2 17222.867} C_VEL
LIN {X 0,Y 355.373,Z 781.775,A -85,B 0,C 180,E1 17220.053,E2 17220.053} C_VEL
LIN {X 0,Y 351.976,Z 795.68,A -85,B 0,C 180,E1 17217.033,E2 17217.033} C_VEL
LIN {X 0,Y 349.161,Z 808.139,A -85,B 0,C 180,E1 17213.813,E2 17213.813} C_VEL
LIN {X 0,Y 347.078,Z 818.664,A -85,B 0,C 180,E1 17210.569,E2 17210.569} C_VEL
LIN {X 0,Y 345.567,Z 827.752,A -85,B 0,C 180,E1 17207.165,E2 17207.165} C_VEL
LIN {X 0,Y 344.644,Z 834.986,A -85,B 0,C 180,E1 17203.762,E2 17203.762} C_VEL
LIN {X 0,Y 344.185,Z 840.619,A -85,B 0,C 180,E1 17200.376,E2 17200.376} C_VEL
LIN {X 0,Y 344.039,Z 844.414,A -85,B 0,C 180,E1 17197.179,E2 17197.179} C_VEL
LIN {X 0,Y 344.012,Z 846.947,A -85,B 0,C 180,E1 17193.833,E2 17193.833} C_VEL
LIN {X 0,Y 344.03,Z 847.884,A -85,B 0,C 180,E1 17190.833,E2 17190.833} C_VEL
LIN {X 0,Y 344.02,Z 847.531,A -85,B 0,C 180,E1 17187.501,E2 17187.501} C_VEL
LIN {X 0,Y 344.015,Z 845.731,A -85,B 0,C 180,E1 17184.329,E2 17184.329} C_VEL
LIN {X 0,Y 344.102,Z 842.16,A -85,B 0,C 180,E1 17180.804,E2 17180.804} C_VEL
LIN {X 0,Y 344.416,Z 837.448,A -85,B 0,C 180,E1 17177.595,E2 17177.595} C_VEL
LIN {X 0,Y 345.166,Z 830.592,A -85,B 0,C 180,E1 17174.094,E2 17174.094} C_VEL
LIN {X 0,Y 346.473,Z 822.024,A -85,B 0,C 180,E1 17170.618,E2 17170.618} C_VEL
LIN {X 0,Y 348.32,Z 812.249,A -85,B 0,C 180,E1 17167.379,E2 17167.379} C_VEL
LIN {X 0,Y 350.856,Z 800.493,A -85,B 0,C 180,E1 17164.151,E2 17164.151} C_VEL
LIN {X 0,Y 354.155,Z 786.577,A -85,B 0,C 180,E1 17160.949,E2 17160.949} C_VEL
LIN {X 0,Y 357.796,Z 771.978,A -85,B 0,C 180,E1 17158.12,E2 17158.12} C_VEL
LIN {X 0,Y 361.869,Z 755.906,A -85,B 0,C 180,E1 17155.5,E2 17155.5} C_VEL
LIN {X 0,Y 366.108,Z 738.718,A -85,B 0,C 180,E1 17153.148,E2 17153.148} C_VEL
LIN {X 0,Y 370.561,Z 719.943,A -85,B 0,C 180,E1 17150.994,E2 17150.994} C_VEL
LIN {X 0,Y 374.774,Z 700.999,A -85,B 0,C 180,E1 17149.185,E2 17149.185} C_VEL
LIN {X 0,Y 378.827,Z 680.673,A -85,B 0,C 180,E1 17147.597,E2 17147.597} C_VEL
LIN {X 0,Y 382.332,Z 660.552,A -85,B 0,C 180,E1 17146.34,E2 17146.34} C_VEL
LIN {X 0,Y 385.541,Z 638.629,A -85,B 0,C 180,E1 17145.262,E2 17145.262} C_VEL
LIN {X 0,Y 388.024,Z 617.489,A -85,B 0,C 180,E1 17144.487,E2 17144.487} C_VEL
LIN {X 0,Y 389.731,Z 594.759,A -85,B 0,C 180,E1 17143.909,E2 17143.909} C_VEL
LIN {X 0,Y 399.987,Z 375.705,A -85,B 0,C 180,E1 17139.526,E2 17139.526} C_VEL
LIN {X 0,Y 400.159,Z 369.051,A -85,B 0,C 180,E1 17139.371,E2 17139.371} C_VEL
LIN {X 0,Y 390.135,Z 352.345,A -85,B 0,C 180,E1 17137.216,E2 17137.216} C_VEL
LIN {X 0,Y 380.264,Z 337.338,A -85,B 0,C 180,E1 17134.928,E2 17134.928} C_VEL
LIN {X 0,Y 370.966,Z 324.261,A -85,B 0,C 180,E1 17132.573,E2 17132.573} C_VEL
LIN {X 0,Y 363.464,Z 314.404,A -85,B 0,C 180,E1 17130.5,E2 17130.5} C_VEL
LIN {X 0,Y 360.011,Z 309.752,A -85,B 0,C 180,E1 17129.444,E2 17129.444} C_VEL
LIN {X 0,Y 356.984,Z 304.516,A -85,B 0,C 180,E1 17127.706,E2 17127.706} C_VEL
LIN {X 0,Y 354.498,Z 299.938,A -85,B 0,C 180,E1 17126.103,E2 17126.103} C_VEL
LIN {X 0,Y 352.358,Z 296.125,A -85,B 0,C 180,E1 17124.653,E2 17124.653} C_VEL
LIN {X 0,Y 349.56,Z 291.616,A -85,B 0,C 180,E1 17122.714,E2 17122.714} C_VEL
LIN {X 0,Y 348.8,Z 289.955,A -85,B 0,C 180,E1 17122.056,E2 17122.056} C_VEL
LIN {X 0,Y 346.319,Z 286.439,A -85,B 0,C 180,E1 17120.235,E2 17120.235} C_VEL
LIN {X 0,Y 345.892,Z 284.798,A -85,B 0,C 180,E1 17119.416,E2 17119.416} C_VEL
LIN {X 0,Y 345.869,Z 284.628,A -85,B 0,C 180,E1 17115.252,E2 17115.252} C_VEL
LIN {X 0,Y 345.871,Z 284.628,A -85,B 0,C 180,E1 17111.168,E2 17111.168} C_VEL
LIN {X 0,Y 345.887,Z 284.626,A -85,B 0,C 180,E1 17106.973,E2 17106.973} C_VEL
LIN {X 0,Y 345.897,Z 284.625,A -85,B 0,C 180,E1 17102.816,E2 17102.816} C_VEL
LIN {X 0,Y 345.913,Z 284.623,A -85,B 0,C 180,E1 17098.675,E2 17098.675} C_VEL
LIN {X 0,Y 345.911,Z 284.622,A -85,B 0,C 180,E1 17094.36,E2 17094.36} C_VEL
LIN {X 0,Y 345.906,Z 284.624,A -85,B 0,C 180,E1 17090.18,E2 17090.18} C_VEL
LIN {X 0,Y 345.901,Z 284.626,A -85,B 0,C 180,E1 17085.947,E2 17085.947} C_VEL
LIN {X 0,Y 345.903,Z 284.627,A -85,B 0,C 180,E1 17081.809,E2 17081.809} C_VEL
LIN {X 0,Y 345.913,Z 284.708,A -85,B 0,C 180,E1 17077.57,E2 17077.57} C_VEL
LIN {X 0,Y 345.984,Z 285.109,A -85,B 0,C 180,E1 17077.037,E2 17077.037} C_VEL
LIN {X 0,Y 347.72,Z 288.801,A -85,B 0,C 180,E1 17075.316,E2 17075.316} C_VEL
LIN {X 0,Y 349.103,Z 290.497,A -85,B 0,C 180,E1 17074.375,E2 17074.375} C_VEL
LIN {X 0,Y 350.922,Z 294.142,A -85,B 0,C 180,E1 17072.878,E2 17072.878} C_VEL
LIN {X 0,Y 352.139,Z 295.959,A -85,B 0,C 180,E1 17072.063,E2 17072.063} C_VEL
LIN {X 0,Y 354.257,Z 299.705,A -85,B 0,C 180,E1 17070.587,E2 17070.587} C_VEL
LIN {X 0,Y 357.659,Z 306.225,A -85,B 0,C 180,E1 17068.293,E2 17068.293} C_VEL
LIN {X 0,Y 360.499,Z 311.798,A -85,B 0,C 180,E1 17066.5,E2 17066.5} C_VEL
LIN {X 0,Y 364.164,Z 318.898,A -85,B 0,C 180,E1 17064.359,E2 17064.359} C_VEL
LIN {X 0,Y 366.194,Z 322.615,A -85,B 0,C 180,E1 17063.422,E2 17063.422} C_VEL
LIN {X 0,Y 376.645,Z 337.766,A -85,B 0,C 180,E1 17060.669,E2 17060.669} C_VEL
LIN {X 0,Y 386.913,Z 353.633,A -85,B 0,C 180,E1 17058.235,E2 17058.235} C_VEL
LIN {X 0,Y 396.974,Z 371.029,A -85,B 0,C 180,E1 17056.035,E2 17056.035} C_VEL
LIN {X 0,Y 397.552,Z 376.881,A -85,B 0,C 180,E1 17055.791,E2 17055.791} C_VEL
LIN {X 0,Y 388.883,Z 595.845,A -85,B 0,C 180,E1 17051.714,E2 17051.714} C_VEL
LIN {X 0,Y 387.054,Z 616.843,A -85,B 0,C 180,E1 17051.085,E2 17051.085} C_VEL
LIN {X 0,Y 384.601,Z 636.624,A -85,B 0,C 180,E1 17050.242,E2 17050.242} C_VEL
LIN {X 0,Y 381.425,Z 656.702,A -85,B 0,C 180,E1 17049.11,E2 17049.11} C_VEL
LIN {X 0,Y 377.869,Z 675.366,A -85,B 0,C 180,E1 17047.774,E2 17047.774} C_VEL
LIN {X 0,Y 374.017,Z 692.941,A -85,B 0,C 180,E1 17046.213,E2 17046.213} C_VEL
LIN {X 0,Y 369.876,Z 709.649,A -85,B 0,C 180,E1 17044.399,E2 17044.399} C_VEL
LIN {X 0,Y 365.458,Z 726.103,A -85,B 0,C 180,E1 17042.241,E2 17042.241} C_VEL
LIN {X 0,Y 361.228,Z 740.998,A -85,B 0,C 180,E1 17039.882,E2 17039.882} C_VEL
LIN {X 0,Y 357.293,Z 754.48,A -85,B 0,C 180,E1 17037.318,E2 17037.318} C_VEL
LIN {X 0,Y 353.557,Z 767.195,A -85,B 0,C 180,E1 17034.386,E2 17034.386} C_VEL
LIN {X 0,Y 350.4,Z 778.263,A -85,B 0,C 180,E1 17031.246,E2 17031.246} C_VEL
LIN {X 0,Y 347.999,Z 787.326,A -85,B 0,C 180,E1 17028.077,E2 17028.077} C_VEL
LIN {X 0,Y 346.185,Z 795.16,A -85,B 0,C 180,E1 17024.634,E2 17024.634} C_VEL
LIN {X 0,Y 345.052,Z 801.143,A -85,B 0,C 180,E1 17021.195,E2 17021.195} C_VEL
LIN {X 0,Y 344.457,Z 805.38,A -85,B 0,C 180,E1 17017.841,E2 17017.841} C_VEL
LIN {X 0,Y 344.178,Z 808.114,A -85,B 0,C 180,E1 17014.332,E2 17014.332} C_VEL
LIN {X 0,Y 344.104,Z 809.251,A -85,B 0,C 180,E1 17010.999,E2 17010.999} C_VEL
LIN {X 0,Y 344.099,Z 809.287,A -85,B 0,C 180,E1 17010.713,E2 17010.713} C_VEL
LIN {X 0,Y 343.094,Z 809.402,A -85,B 0,C 180,E1 17009.431,E2 17009.431} C_VEL
LIN {X 0,Y 338.683,Z 809.162,A -85,B 0,C 180,E1 17007.096,E2 17007.096} C_VEL
LIN {X 0,Y 336.404,Z 808.54,A -85,B 0,C 180,E1 17005.429,E2 17005.429} C_VEL
LIN {X 0,Y 336.229,Z 808.193,A -85,B 0,C 180,E1 17004.861,E2 17004.861} C_VEL
LIN {X 0,Y 336.587,Z 805.183,A -85,B 0,C 180,E1 17001.286,E2 17001.286} C_VEL
LIN {X 0,Y 337.315,Z 800.775,A -85,B 0,C 180,E1 16997.851,E2 16997.851} C_VEL
LIN {X 0,Y 338.688,Z 794.307,A -85,B 0,C 180,E1 16994.24,E2 16994.24} C_VEL
LIN {X 0,Y 340.719,Z 786.307,A -85,B 0,C 180,E1 16990.812,E2 16990.812} C_VEL
LIN {X 0,Y 343.412,Z 776.867,A -85,B 0,C 180,E1 16987.579,E2 16987.579} C_VEL
LIN {X 0,Y 346.774,Z 765.79,A -85,B 0,C 180,E1 16984.486,E2 16984.486} C_VEL
LIN {X 0,Y 350.494,Z 753.885,A -85,B 0,C 180,E1 16981.736,E2 16981.736} C_VEL
LIN {X 0,Y 354.98,Z 739.333,A -85,B 0,C 180,E1 16978.974,E2 16978.974} C_VEL
LIN {X 0,Y 359.486,Z 724.018,A -85,B 0,C 180,E1 16976.585,E2 16976.585} C_VEL
LIN {X 0,Y 363.996,Z 707.703,A -85,B 0,C 180,E1 16974.483,E2 16974.483} C_VEL
LIN {X 0,Y 368.541,Z 689.691,A -85,B 0,C 180,E1 16972.577,E2 16972.577} C_VEL
LIN {X 0,Y 372.662,Z 671.269,A -85,B 0,C 180,E1 16970.994,E2 16970.994} C_VEL
LIN {X 0,Y 376.297,Z 652.408,A -85,B 0,C 180,E1 16969.693,E2 16969.693} C_VEL
LIN {X 0,Y 379.363,Z 632.57,A -85,B 0,C 180,E1 16968.634,E2 16968.634} C_VEL
LIN {X 0,Y 381.774,Z 612.281,A -85,B 0,C 180,E1 16967.829,E2 16967.829} C_VEL
LIN {X 0,Y 383.503,Z 590.595,A -85,B 0,C 180,E1 16967.242,E2 16967.242} C_VEL
LIN {X 0,Y 392.271,Z 376.859,A -85,B 0,C 180,E1 16963.222,E2 16963.222} C_VEL
LIN {X 0,Y 391.776,Z 374.667,A -85,B 0,C 180,E1 16963.08,E2 16963.08} C_VEL
LIN {X 0,Y 381.427,Z 356.952,A -85,B 0,C 180,E1 16960.723,E2 16960.723} C_VEL
LIN {X 0,Y 370.985,Z 340.655,A -85,B 0,C 180,E1 16958.111,E2 16958.111} C_VEL
LIN {X 0,Y 361.558,Z 327.172,A -85,B 0,C 180,E1 16955.503,E2 16955.503} C_VEL
LIN {X 0,Y 356.799,Z 320.297,A -85,B 0,C 180,E1 16953.957,E2 16953.957} C_VEL
LIN {X 0,Y 351.854,Z 310.57,A -85,B 0,C 180,E1 16950.764,E2 16950.764} C_VEL
LIN {X 0,Y 348.915,Z 305.333,A -85,B 0,C 180,E1 16948.779,E2 16948.779} C_VEL
LIN {X 0,Y 346.709,Z 301.111,A -85,B 0,C 180,E1 16947.107,E2 16947.107} C_VEL
LIN {X 0,Y 344.541,Z 297.371,A -85,B 0,C 180,E1 16945.436,E2 16945.436} C_VEL
LIN {X 0,Y 343.724,Z 295.936,A -85,B 0,C 180,E1 16944.764,E2 16944.764} C_VEL
LIN {X 0,Y 341.543,Z 292.299,A -85,B 0,C 180,E1 16942.915,E2 16942.915} C_VEL
LIN {X 0,Y 340.644,Z 290.688,A -85,B 0,C 180,E1 16942.068,E2 16942.068} C_VEL
LIN {X 0,Y 338.428,Z 287.455,A -85,B 0,C 180,E1 16940.036,E2 16940.036} C_VEL
LIN {X 0,Y 337.992,Z 285.765,A -85,B 0,C 180,E1 16938.99,E2 16938.99} C_VEL
LIN {X 0,Y 337.956,Z 285.614,A -85,B 0,C 180,E1 16934.666,E2 16934.666} C_VEL
LIN {X 0,Y 337.952,Z 285.613,A -85,B 0,C 180,E1 16930.398,E2 16930.398} C_VEL
LIN {X 0,Y 337.951,Z 285.613,A -85,B 0,C 180,E1 16926.114,E2 16926.114} C_VEL
LIN {X 0,Y 337.954,Z 285.614,A -85,B 0,C 180,E1 16921.865,E2 16921.865} C_VEL
LIN {X 0,Y 337.95,Z 285.617,A -85,B 0,C 180,E1 16917.796,E2 16917.796} C_VEL
LIN {X 0,Y 337.961,Z 285.617,A -85,B 0,C 180,E1 16913.545,E2 16913.545} C_VEL
LIN {X 0,Y 337.955,Z 285.616,A -85,B 0,C 180,E1 16909.258,E2 16909.258} C_VEL
LIN {X 0,Y 337.953,Z 285.616,A -85,B 0,C 180,E1 16905.085,E2 16905.085} C_VEL
LIN {X 0,Y 338.007,Z 286.158,A -85,B 0,C 180,E1 16903.856,E2 16903.856} C_VEL
LIN {X 0,Y 339.76,Z 289.807,A -85,B 0,C 180,E1 16901.824,E2 16901.824} C_VEL
LIN {X 0,Y 341.365,Z 291.695,A -85,B 0,C 180,E1 16900.581,E2 16900.581} C_VEL
LIN {X 0,Y 343.59,Z 295.795,A -85,B 0,C 180,E1 16898.62,E2 16898.62} C_VEL
LIN {X 0,Y 344.681,Z 297.281,A -85,B 0,C 180,E1 16897.846,E2 16897.846} C_VEL
LIN {X 0,Y 346.819,Z 301.168,A -85,B 0,C 180,E1 16896.196,E2 16896.196} C_VEL
LIN {X 0,Y 347.736,Z 302.763,A -85,B 0,C 180,E1 16895.541,E2 16895.541} C_VEL
LIN {X 0,Y 350.596,Z 307.932,A -85,B 0,C 180,E1 16893.568,E2 16893.568} C_VEL
LIN {X 0,Y 352.508,Z 311.034,A -85,B 0,C 180,E1 16892.536,E2 16892.536} C_VEL
LIN {X 0,Y 358.425,Z 318.513,A -85,B 0,C 180,E1 16890.642,E2 16890.642} C_VEL
LIN {X 0,Y 365.698,Z 327.979,A -85,B 0,C 180,E1 16888.519,E2 16888.519} C_VEL
LIN {X 0,Y 375.37,Z 341.686,A -85,B 0,C 180,E1 16885.942,E2 16885.942} C_VEL
LIN {X 0,Y 385.232,Z 356.702,A -85,B 0,C 180,E1 16883.556,E2 16883.556} C_VEL
LIN {X 0,Y 394.862,Z 372.864,A -85,B 0,C 180,E1 16881.403,E2 16881.403} C_VEL
LIN {X 0,Y 384.163,Z 592.433,A -85,B 0,C 180,E1 16876.978,E2 16876.978} C_VEL
LIN {X 0,Y 382.452,Z 615.113,A -85,B 0,C 180,E1 16876.411,E2 16876.411} C_VEL
LIN {X 0,Y 379.93,Z 636.614,A -85,B 0,C 180,E1 16875.644,E2 16875.644} C_VEL
LIN {X 0,Y 376.91,Z 657.145,A -85,B 0,C 180,E1 16874.665,E2 16874.665} C_VEL
LIN {X 0,Y 373.462,Z 676.651,A -85,B 0,C 180,E1 16873.475,E2 16873.475} C_VEL
LIN {X 0,Y 369.361,Z 696.66,A -85,B 0,C 180,E1 16871.96,E2 16871.96} C_VEL
LIN {X 0,Y 364.799,Z 716.727,A -85,B 0,C 180,E1 16870.097,E2 16870.097} C_VEL
LIN {X 0,Y 360.315,Z 735.157,A -85,B 0,C 180,E1 16868.026,E2 16868.026} C_VEL
LIN {X 0,Y 355.793,Z 752.441,A -85,B 0,C 180,E1 16865.694,E2 16865.694} C_VEL
LIN {X 0,Y 351.511,Z 768.561,A -85,B 0,C 180,E1 16863.101,E2 16863.101} C_VEL
LIN {X 0,Y 347.518,Z 783.648,A -85,B 0,C 180,E1 16860.231,E2 16860.231} C_VEL
LIN {X 0,Y 344.047,Z 797.323,A -85,B 0,C 180,E1 16857.146,E2 16857.146} C_VEL
LIN {X 0,Y 341.166,Z 809.429,A -85,B 0,C 180,E1 16853.855,E2 16853.855} C_VEL
LIN {X 0,Y 339.044,Z 819.6,A -85,B 0,C 180,E1 16850.544,E2 16850.544} C_VEL
LIN {X 0,Y 337.518,Z 828.468,A -85,B 0,C 180,E1 16847.054,E2 16847.054} C_VEL
LIN {X 0,Y 336.602,Z 835.477,A -85,B 0,C 180,E1 16843.571,E2 16843.571} C_VEL
LIN {X 0,Y 336.163,Z 840.825,A -85,B 0,C 180,E1 16840.102,E2 16840.102} C_VEL
LIN {X 0,Y 336.025,Z 844.64,A -85,B 0,C 180,E1 16836.664,E2 16836.664} C_VEL
LIN {X 0,Y 336.029,Z 846.718,A -85,B 0,C 180,E1 16833.412,E2 16833.412} C_VEL
LIN {X 0,Y 336.045,Z 847.531,A -85,B 0,C 180,E1 16830.17,E2 16830.17} C_VEL
LIN {X 0,Y 336.03,Z 846.789,A -85,B 0,C 180,E1 16826.759,E2 16826.759} C_VEL
LIN {X 0,Y 336.02,Z 844.783,A -85,B 0,C 180,E1 16823.508,E2 16823.508} C_VEL
LIN {X 0,Y 336.152,Z 841.034,A -85,B 0,C 180,E1 16820.066,E2 16820.066} C_VEL
LIN {X 0,Y 336.572,Z 835.793,A -85,B 0,C 180,E1 16816.602,E2 16816.602} C_VEL
LIN {X 0,Y 337.458,Z 828.833,A -85,B 0,C 180,E1 16813.121,E2 16813.121} C_VEL
LIN {X 0,Y 338.947,Z 820.069,A -85,B 0,C 180,E1 16809.63,E2 16809.63} C_VEL
LIN {X 0,Y 341.036,Z 810.013,A -85,B 0,C 180,E1 16806.319,E2 16806.319} C_VEL
LIN {X 0,Y 343.872,Z 797.969,A -85,B 0,C 180,E1 16803.026,E2 16803.026} C_VEL
LIN {X 0,Y 347.301,Z 784.42,A -85,B 0,C 180,E1 16799.939,E2 16799.939} C_VEL
LIN {X 0,Y 351.38,Z 769.001,A -85,B 0,C 180,E1 16796.982,E2 16796.982} C_VEL
LIN {X 0,Y 355.606,Z 753.102,A -85,B 0,C 180,E1 16794.408,E2 16794.408} C_VEL
LIN {X 0,Y 360.177,Z 735.58,A -85,B 0,C 180,E1 16792.035,E2 16792.035} C_VEL
LIN {X 0,Y 364.609,Z 717.403,A -85,B 0,C 180,E1 16789.981,E2 16789.981} C_VEL
LIN {X 0,Y 369.133,Z 697.57,A -85,B 0,C 180,E1 16788.123,E2 16788.123} C_VEL
LIN {X 0,Y 373.241,Z 677.659,A -85,B 0,C 180,E1 16786.598,E2 16786.598} C_VEL
LIN {X 0,Y 376.679,Z 658.287,A -85,B 0,C 180,E1 16785.407,E2 16785.407} C_VEL
LIN {X 0,Y 379.866,Z 636.824,A -85,B 0,C 180,E1 16784.372,E2 16784.372} C_VEL
LIN {X 0,Y 382.394,Z 615.292,A -85,B 0,C 180,E1 16783.601,E2 16783.601} C_VEL
LIN {X 0,Y 384.112,Z 592.517,A -85,B 0,C 180,E1 16783.031,E2 16783.031} C_VEL
LIN {X 0,Y 394.776,Z 373.37,A -85,B 0,C 180,E1 16778.614,E2 16778.614} C_VEL
LIN {X 0,Y 394.461,Z 372.191,A -85,B 0,C 180,E1 16778.529,E2 16778.529} C_VEL
LIN {X 0,Y 384.164,Z 355.02,A -85,B 0,C 180,E1 16776.214,E2 16776.214} C_VEL
LIN {X 0,Y 373.501,Z 338.943,A -85,B 0,C 180,E1 16773.605,E2 16773.605} C_VEL
LIN {X 0,Y 364.013,Z 325.863,A -85,B 0,C 180,E1 16771.044,E2 16771.044} C_VEL
LIN {X 0,Y 360.071,Z 320.709,A -85,B 0,C 180,E1 16769.897,E2 16769.897} C_VEL
LIN {X 0,Y 356.253,Z 315.774,A -85,B 0,C 180,E1 16768.726,E2 16768.726} C_VEL
LIN {X 0,Y 351.772,Z 310.139,A -85,B 0,C 180,E1 16767.233,E2 16767.233} C_VEL
LIN {X 0,Y 349.535,Z 306.004,A -85,B 0,C 180,E1 16765.772,E2 16765.772} C_VEL
LIN {X 0,Y 347,Z 301.368,A -85,B 0,C 180,E1 16763.971,E2 16763.971} C_VEL
LIN {X 0,Y 344.768,Z 297.584,A -85,B 0,C 180,E1 16762.328,E2 16762.328} C_VEL
LIN {X 0,Y 343.922,Z 296.145,A -85,B 0,C 180,E1 16761.667,E2 16761.667} C_VEL
LIN {X 0,Y 341.652,Z 292.526,A -85,B 0,C 180,E1 16759.845,E2 16759.845} C_VEL
LIN {X 0,Y 340.769,Z 290.819,A -85,B 0,C 180,E1 16759.007,E2 16759.007} C_VEL
LIN {X 0,Y 338.462,Z 287.618,A -85,B 0,C 180,E1 16757.005,E2 16757.005} C_VEL
LIN {X 0,Y 337.946,Z 285.814,A -85,B 0,C 180,E1 16755.944,E2 16755.944} C_VEL
LIN {X 0,Y 337.92,Z 285.618,A -85,B 0,C 180,E1 16751.953,E2 16751.953} C_VEL
LIN {X 0,Y 337.923,Z 285.618,A -85,B 0,C 180,E1 16747.615,E2 16747.615} C_VEL
LIN {X 0,Y 337.933,Z 285.617,A -85,B 0,C 180,E1 16743.392,E2 16743.392} C_VEL
LIN {X 0,Y 337.938,Z 285.619,A -85,B 0,C 180,E1 16739.322,E2 16739.322} C_VEL
LIN {X 0,Y 337.953,Z 285.619,A -85,B 0,C 180,E1 16735.078,E2 16735.078} C_VEL
LIN {X 0,Y 337.961,Z 285.622,A -85,B 0,C 180,E1 16730.978,E2 16730.978} C_VEL
LIN {X 0,Y 337.982,Z 285.62,A -85,B 0,C 180,E1 16726.658,E2 16726.658} C_VEL
LIN {X 0,Y 337.987,Z 285.618,A -85,B 0,C 180,E1 16722.437,E2 16722.437} C_VEL
LIN {X 0,Y 338.048,Z 286.02,A -85,B 0,C 180,E1 16720.497,E2 16720.497} C_VEL
LIN {X 0,Y 339.577,Z 289.494,A -85,B 0,C 180,E1 16718.585,E2 16718.585} C_VEL
LIN {X 0,Y 341.405,Z 291.909,A -85,B 0,C 180,E1 16717.076,E2 16717.076} C_VEL
LIN {X 0,Y 343.496,Z 295.7,A -85,B 0,C 180,E1 16715.218,E2 16715.218} C_VEL
LIN {X 0,Y 344.416,Z 297.032,A -85,B 0,C 180,E1 16714.532,E2 16714.532} C_VEL
LIN {X 0,Y 346.485,Z 300.858,A -85,B 0,C 180,E1 16712.874,E2 16712.874} C_VEL
LIN {X 0,Y 347.563,Z 302.943,A -85,B 0,C 180,E1 16712.036,E2 16712.036} C_VEL
LIN {X 0,Y 349.954,Z 307.086,A -85,B 0,C 180,E1 16710.377,E2 16710.377} C_VEL
LIN {X 0,Y 352.834,Z 312.755,A -85,B 0,C 180,E1 16708.382,E2 16708.382} C_VEL
LIN {X 0,Y 356.811,Z 320.335,A -85,B 0,C 180,E1 16705.913,E2 16705.913} C_VEL
LIN {X 0,Y 360.396,Z 325.642,A -85,B 0,C 180,E1 16704.707,E2 16704.707} C_VEL
LIN {X 0,Y 369.065,Z 337.884,A -85,B 0,C 180,E1 16702.271,E2 16702.271} C_VEL
LIN {X 0,Y 379.63,Z 354.085,A -85,B 0,C 180,E1 16699.588,E2 16699.588} C_VEL
LIN {X 0,Y 389.481,Z 370.736,A -85,B 0,C 180,E1 16697.308,E2 16697.308} C_VEL
LIN {X 0,Y 392.056,Z 375.69,A -85,B 0,C 180,E1 16696.733,E2 16696.733} C_VEL
LIN {X 0,Y 392.137,Z 379.828,A -85,B 0,C 180,E1 16696.611,E2 16696.611} C_VEL
LIN {X 0,Y 383.155,Z 595.929,A -85,B 0,C 180,E1 16692.546,E2 16692.546} C_VEL
LIN {X 0,Y 381.257,Z 616.924,A -85,B 0,C 180,E1 16691.912,E2 16691.912} C_VEL
LIN {X 0,Y 378.79,Z 636.191,A -85,B 0,C 180,E1 16691.09,E2 16691.09} C_VEL
LIN {X 0,Y 375.642,Z 655.641,A -85,B 0,C 180,E1 16690,E2 16690} C_VEL
LIN {X 0,Y 371.996,Z 674.314,A -85,B 0,C 180,E1 16688.675,E2 16688.675} C_VEL
LIN {X 0,Y 367.835,Z 692.541,A -85,B 0,C 180,E1 16687.053,E2 16687.053} C_VEL
LIN {X 0,Y 363.532,Z 709.314,A -85,B 0,C 180,E1 16685.227,E2 16685.227} C_VEL
LIN {X 0,Y 358.986,Z 725.591,A -85,B 0,C 180,E1 16683.085,E2 16683.085} C_VEL
LIN {X 0,Y 354.819,Z 739.739,A -85,B 0,C 180,E1 16680.854,E2 16680.854} C_VEL
LIN {X 0,Y 350.481,Z 753.84,A -85,B 0,C 180,E1 16678.173,E2 16678.173} C_VEL
LIN {X 0,Y 346.586,Z 766.353,A -85,B 0,C 180,E1 16675.274,E2 16675.274} C_VEL
LIN {X 0,Y 343.325,Z 777.107,A -85,B 0,C 180,E1 16672.246,E2 16672.246} C_VEL
LIN {X 0,Y 340.535,Z 786.93,A -85,B 0,C 180,E1 16668.842,E2 16668.842} C_VEL
LIN {X 0,Y 338.563,Z 794.784,A -85,B 0,C 180,E1 16665.414,E2 16665.414} C_VEL
LIN {X 0,Y 337.288,Z 800.896,A -85,B 0,C 180,E1 16661.969,E2 16661.969} C_VEL
LIN {X 0,Y 336.548,Z 805.455,A -85,B 0,C 180,E1 16658.37,E2 16658.37} C_VEL
LIN {X 0,Y 336.224,Z 808.247,A -85,B 0,C 180,E1 16654.947,E2 16654.947} C_VEL
LIN {X 0,Y 336.114,Z 809.657,A -85,B 0,C 180,E1 16651.364,E2 16651.364} C_VEL
LIN {X 0,Y 336.125,Z 809.586,A -85,B 0,C 180,E1 16647.954,E2 16647.954} C_VEL
LIN {X 0,Y 336.229,Z 808.193,A -85,B 0,C 180,E1 16644.861,E2 16644.861} C_VEL
LIN {X 0,Y 335.323,Z 807.383,A -85,B 0,C 180,E1 16643.553,E2 16643.553} C_VEL
LIN {X 0,Y 329.471,Z 804.383,A -85,B 0,C 180,E1 16639.958,E2 16639.958} C_VEL
LIN {X 0,Y 329.06,Z 803.087,A -85,B 0,C 180,E1 16638.916,E2 16638.916} C_VEL
LIN {X 0,Y 330.179,Z 797.778,A -85,B 0,C 180,E1 16635.443,E2 16635.443} C_VEL
LIN {X 0,Y 332.117,Z 790.239,A -85,B 0,C 180,E1 16631.754,E2 16631.754} C_VEL
LIN {X 0,Y 334.631,Z 781.563,A -85,B 0,C 180,E1 16628.438,E2 16628.438} C_VEL
LIN {X 0,Y 337.756,Z 771.585,A -85,B 0,C 180,E1 16625.33,E2 16625.33} C_VEL
LIN {X 0,Y 341.661,Z 759.621,A -85,B 0,C 180,E1 16622.271,E2 16622.271} C_VEL
LIN {X 0,Y 345.784,Z 747.032,A -85,B 0,C 180,E1 16619.602,E2 16619.602} C_VEL
LIN {X 0,Y 350.538,Z 732.037,A -85,B 0,C 180,E1 16616.99,E2 16616.99} C_VEL
LIN {X 0,Y 355.175,Z 716.481,A -85,B 0,C 180,E1 16614.754,E2 16614.754} C_VEL
LIN {X 0,Y 359.912,Z 699.38,A -85,B 0,C 180,E1 16612.728,E2 16612.728} C_VEL
LIN {X 0,Y 364.408,Z 681.275,A -85,B 0,C 180,E1 16610.973,E2 16610.973} C_VEL
LIN {X 0,Y 368.353,Z 663.246,A -85,B 0,C 180,E1 16609.555,E2 16609.555} C_VEL
LIN {X 0,Y 371.787,Z 644.282,A -85,B 0,C 180,E1 16608.375,E2 16608.375} C_VEL
LIN {X 0,Y 374.685,Z 624.507,A -85,B 0,C 180,E1 16607.431,E2 16607.431} C_VEL
LIN {X 0,Y 376.966,Z 603.266,A -85,B 0,C 180,E1 16606.696,E2 16606.696} C_VEL
LIN {X 0,Y 378.354,Z 581.299,A -85,B 0,C 180,E1 16606.193,E2 16606.193} C_VEL
LIN {X 0,Y 386.957,Z 379.139,A -85,B 0,C 180,E1 16602.363,E2 16602.363} C_VEL
LIN {X 0,Y 377.385,Z 362.553,A -85,B 0,C 180,E1 16600.102,E2 16600.102} C_VEL
LIN {X 0,Y 367.631,Z 347.071,A -85,B 0,C 180,E1 16597.583,E2 16597.583} C_VEL
LIN {X 0,Y 358.36,Z 333.61,A -85,B 0,C 180,E1 16594.937,E2 16594.937} C_VEL
LIN {X 0,Y 352.146,Z 325.226,A -85,B 0,C 180,E1 16592.987,E2 16592.987} C_VEL
LIN {X 0,Y 348.488,Z 320.082,A -85,B 0,C 180,E1 16591.672,E2 16591.672} C_VEL
LIN {X 0,Y 346.285,Z 315.778,A -85,B 0,C 180,E1 16590.16,E2 16590.16} C_VEL
LIN {X 0,Y 344.194,Z 311.74,A -85,B 0,C 180,E1 16588.641,E2 16588.641} C_VEL
LIN {X 0,Y 341.758,Z 307.217,A -85,B 0,C 180,E1 16586.779,E2 16586.779} C_VEL
LIN {X 0,Y 339.066,Z 302.364,A -85,B 0,C 180,E1 16584.569,E2 16584.569} C_VEL
LIN {X 0,Y 336.879,Z 298.574,A -85,B 0,C 180,E1 16582.628,E2 16582.628} C_VEL
LIN {X 0,Y 335.828,Z 296.9,A -85,B 0,C 180,E1 16581.666,E2 16581.666} C_VEL
LIN {X 0,Y 333.794,Z 293.528,A -85,B 0,C 180,E1 16579.603,E2 16579.603} C_VEL
LIN {X 0,Y 333.109,Z 292.053,A -85,B 0,C 180,E1 16578.734,E2 16578.734} C_VEL
LIN {X 0,Y 330.522,Z 288.511,A -85,B 0,C 180,E1 16575.799,E2 16575.799} C_VEL
LIN {X 0,Y 330.04,Z 286.769,A -85,B 0,C 180,E1 16574.384,E2 16574.384} C_VEL
LIN {X 0,Y 330.02,Z 286.6,A -85,B 0,C 180,E1 16570.062,E2 16570.062} C_VEL
LIN {X 0,Y 330.019,Z 286.6,A -85,B 0,C 180,E1 16565.913,E2 16565.913} C_VEL
LIN {X 0,Y 330.032,Z 286.599,A -85,B 0,C 180,E1 16561.563,E2 16561.563} C_VEL
LIN {X 0,Y 330.027,Z 286.6,A -85,B 0,C 180,E1 16557.396,E2 16557.396} C_VEL
LIN {X 0,Y 330.014,Z 286.602,A -85,B 0,C 180,E1 16553.04,E2 16553.04} C_VEL
LIN {X 0,Y 330.024,Z 286.825,A -85,B 0,C 180,E1 16548.732,E2 16548.732} C_VEL
LIN {X 0,Y 332.01,Z 290.988,A -85,B 0,C 180,E1 16545.525,E2 16545.525} C_VEL
LIN {X 0,Y 333.591,Z 292.856,A -85,B 0,C 180,E1 16543.994,E2 16543.994} C_VEL
LIN {X 0,Y 335.651,Z 296.736,A -85,B 0,C 180,E1 16541.773,E2 16541.773} C_VEL
LIN {X 0,Y 336.89,Z 298.306,A -85,B 0,C 180,E1 16540.766,E2 16540.766} C_VEL
LIN {X 0,Y 339.17,Z 302.425,A -85,B 0,C 180,E1 16538.741,E2 16538.741} C_VEL
LIN {X 0,Y 340.063,Z 303.72,A -85,B 0,C 180,E1 16538.074,E2 16538.074} C_VEL
LIN {X 0,Y 342.177,Z 307.58,A -85,B 0,C 180,E1 16536.402,E2 16536.402} C_VEL
LIN {X 0,Y 344.442,Z 311.569,A -85,B 0,C 180,E1 16534.925,E2 16534.925} C_VEL
LIN {X 0,Y 347.538,Z 315.331,A -85,B 0,C 180,E1 16533.793,E2 16533.793} C_VEL
LIN {X 0,Y 351.642,Z 320.411,A -85,B 0,C 180,E1 16532.389,E2 16532.389} C_VEL
LIN {X 0,Y 355.685,Z 325.546,A -85,B 0,C 180,E1 16531.086,E2 16531.086} C_VEL
LIN {X 0,Y 362.612,Z 334.687,A -85,B 0,C 180,E1 16529.007,E2 16529.007} C_VEL
LIN {X 0,Y 372.029,Z 348.264,A -85,B 0,C 180,E1 16526.425,E2 16526.425} C_VEL
LIN {X 0,Y 381.466,Z 362.872,A -85,B 0,C 180,E1 16524.073,E2 16524.073} C_VEL
LIN {X 0,Y 389.453,Z 376.527,A -85,B 0,C 180,E1 16522.219,E2 16522.219} C_VEL
LIN {X 0,Y 378.338,Z 595.11,A -85,B 0,C 180,E1 16517.77,E2 16517.77} C_VEL
LIN {X 0,Y 376.5,Z 617.668,A -85,B 0,C 180,E1 16517.184,E2 16517.184} C_VEL
LIN {X 0,Y 373.796,Z 638.972,A -85,B 0,C 180,E1 16516.386,E2 16516.386} C_VEL
LIN {X 0,Y 370.455,Z 660.092,A -85,B 0,C 180,E1 16515.33,E2 16515.33} C_VEL
LIN {X 0,Y 366.679,Z 680.202,A -85,B 0,C 180,E1 16514.052,E2 16514.052} C_VEL
LIN {X 0,Y 362.466,Z 699.581,A -85,B 0,C 180,E1 16512.517,E2 16512.517} C_VEL
LIN {X 0,Y 357.95,Z 718.316,A -85,B 0,C 180,E1 16510.709,E2 16510.709} C_VEL
LIN {X 0,Y 353.407,Z 736.024,A -85,B 0,C 180,E1 16508.661,E2 16508.661} C_VEL
LIN {X 0,Y 348.808,Z 752.847,A -85,B 0,C 180,E1 16506.343,E2 16506.343} C_VEL
LIN {X 0,Y 344.292,Z 768.956,A -85,B 0,C 180,E1 16503.688,E2 16503.688} C_VEL
LIN {X 0,Y 340.11,Z 783.912,A -85,B 0,C 180,E1 16500.765,E2 16500.765} C_VEL
LIN {X 0,Y 336.467,Z 797.471,A -85,B 0,C 180,E1 16497.617,E2 16497.617} C_VEL
LIN {X 0,Y 333.44,Z 809.52,A -85,B 0,C 180,E1 16494.255,E2 16494.255} C_VEL
LIN {X 0,Y 331.203,Z 819.59,A -85,B 0,C 180,E1 16490.868,E2 16490.868} C_VEL
LIN {X 0,Y 329.592,Z 828.362,A -85,B 0,C 180,E1 16487.295,E2 16487.295} C_VEL
LIN {X 0,Y 328.628,Z 835.325,A -85,B 0,C 180,E1 16483.728,E2 16483.728} C_VEL
LIN {X 0,Y 328.17,Z 840.579,A -85,B 0,C 180,E1 16480.178,E2 16480.178} C_VEL
LIN {X 0,Y 328.031,Z 844.336,A -85,B 0,C 180,E1 16476.651,E2 16476.651} C_VEL
LIN {X 0,Y 328.04,Z 846.342,A -85,B 0,C 180,E1 16473.32,E2 16473.32} C_VEL
LIN {X 0,Y 328.062,Z 847.099,A -85,B 0,C 180,E1 16470,E2 16470} C_VEL
LIN {X 0,Y 328.04,Z 846.338,A -85,B 0,C 180,E1 16466.68,E2 16466.68} C_VEL
LIN {X 0,Y 328.03,Z 844.329,A -85,B 0,C 180,E1 16463.349,E2 16463.349} C_VEL
LIN {X 0,Y 328.17,Z 840.57,A -85,B 0,C 180,E1 16459.822,E2 16459.822} C_VEL
LIN {X 0,Y 328.664,Z 834.995,A -85,B 0,C 180,E1 16456.094,E2 16456.094} C_VEL
LIN {X 0,Y 329.658,Z 827.974,A -85,B 0,C 180,E1 16452.527,E2 16452.527} C_VEL
LIN {X 0,Y 331.304,Z 819.087,A -85,B 0,C 180,E1 16448.953,E2 16448.953} C_VEL
LIN {X 0,Y 333.717,Z 808.294,A -85,B 0,C 180,E1 16445.389,E2 16445.389} C_VEL
LIN {X 0,Y 336.835,Z 796.051,A -85,B 0,C 180,E1 16442.031,E2 16442.031} C_VEL
LIN {X 0,Y 340.565,Z 782.271,A -85,B 0,C 180,E1 16438.889,E2 16438.889} C_VEL
LIN {X 0,Y 344.674,Z 767.508,A -85,B 0,C 180,E1 16436.062,E2 16436.062} C_VEL
LIN {X 0,Y 349.29,Z 750.991,A -85,B 0,C 180,E1 16433.395,E2 16433.395} C_VEL
LIN {X 0,Y 353.984,Z 733.81,A -85,B 0,C 180,E1 16431.064,E2 16431.064} C_VEL
LIN {X 0,Y 358.703,Z 715.219,A -85,B 0,C 180,E1 16428.973,E2 16428.973} C_VEL
LIN {X 0,Y 363.278,Z 695.804,A -85,B 0,C 180,E1 16427.172,E2 16427.172} C_VEL
LIN {X 0,Y 367.544,Z 675.636,A -85,B 0,C 180,E1 16425.644,E2 16425.644} C_VEL
LIN {X 0,Y 371.246,Z 655.382,A -85,B 0,C 180,E1 16424.409,E2 16424.409} C_VEL
LIN {X 0,Y 374.434,Z 633.937,A -85,B 0,C 180,E1 16423.409,E2 16423.409} C_VEL
LIN {X 0,Y 377.017,Z 611.615,A -85,B 0,C 180,E1 16422.65,E2 16422.65} C_VEL
LIN {X 0,Y 378.728,Z 586.758,A -85,B 0,C 180,E1 16422.059,E2 16422.059} C_VEL
LIN {X 0,Y 389.392,Z 376.324,A -85,B 0,C 180,E1 16417.785,E2 16417.785} C_VEL
LIN {X 0,Y 379.221,Z 359.289,A -85,B 0,C 180,E1 16415.408,E2 16415.408} C_VEL
LIN {X 0,Y 368.787,Z 343.462,A -85,B 0,C 180,E1 16412.744,E2 16412.744} C_VEL
LIN {X 0,Y 358.254,Z 328.779,A -85,B 0,C 180,E1 16409.741,E2 16409.741} C_VEL
LIN {X 0,Y 352.751,Z 321.857,A -85,B 0,C 180,E1 16408.022,E2 16408.022} C_VEL
LIN {X 0,Y 348.702,Z 316.755,A -85,B 0,C 180,E1 16406.663,E2 16406.663} C_VEL
LIN {X 0,Y 344.813,Z 312.016,A -85,B 0,C 180,E1 16405.276,E2 16405.276} C_VEL
LIN {X 0,Y 343.184,Z 309.542,A -85,B 0,C 180,E1 16404.438,E2 16404.438} C_VEL
LIN {X 0,Y 342.083,Z 307.474,A -85,B 0,C 180,E1 16403.605,E2 16403.605} C_VEL
LIN {X 0,Y 339.315,Z 302.583,A -85,B 0,C 180,E1 16401.431,E2 16401.431} C_VEL
LIN {X 0,Y 336.958,Z 298.521,A -85,B 0,C 180,E1 16399.41,E2 16399.41} C_VEL
LIN {X 0,Y 335.983,Z 297.057,A -85,B 0,C 180,E1 16398.567,E2 16398.567} C_VEL
LIN {X 0,Y 333.981,Z 293.95,A -85,B 0,C 180,E1 16396.669,E2 16396.669} C_VEL
LIN {X 0,Y 333.182,Z 292.159,A -85,B 0,C 180,E1 16395.669,E2 16395.669} C_VEL
LIN {X 0,Y 330.517,Z 288.574,A -85,B 0,C 180,E1 16392.758,E2 16392.758} C_VEL
LIN {X 0,Y 330.013,Z 286.811,A -85,B 0,C 180,E1 16391.357,E2 16391.357} C_VEL
LIN {X 0,Y 329.999,Z 286.603,A -85,B 0,C 180,E1 16387.136,E2 16387.136} C_VEL
LIN {X 0,Y 330.019,Z 286.601,A -85,B 0,C 180,E1 16382.778,E2 16382.778} C_VEL
LIN {X 0,Y 330.034,Z 286.599,A -85,B 0,C 180,E1 16378.611,E2 16378.611} C_VEL
LIN {X 0,Y 330.028,Z 286.599,A -85,B 0,C 180,E1 16374.262,E2 16374.262} C_VEL
LIN {X 0,Y 330.021,Z 286.601,A -85,B 0,C 180,E1 16370.055,E2 16370.055} C_VEL
LIN {X 0,Y 330.027,Z 286.677,A -85,B 0,C 180,E1 16365.794,E2 16365.794} C_VEL
LIN {X 0,Y 330.185,Z 287.402,A -85,B 0,C 180,E1 16364.725,E2 16364.725} C_VEL
LIN {X 0,Y 332.148,Z 291.103,A -85,B 0,C 180,E1 16361.937,E2 16361.937} C_VEL
LIN {X 0,Y 333.552,Z 292.796,A -85,B 0,C 180,E1 16360.565,E2 16360.565} C_VEL
LIN {X 0,Y 335.401,Z 296.427,A -85,B 0,C 180,E1 16358.489,E2 16358.489} C_VEL
LIN {X 0,Y 336.794,Z 298.336,A -85,B 0,C 180,E1 16357.298,E2 16357.298} C_VEL
LIN {X 0,Y 338.842,Z 302.128,A -85,B 0,C 180,E1 16355.413,E2 16355.413} C_VEL
LIN {X 0,Y 339.708,Z 303.449,A -85,B 0,C 180,E1 16354.736,E2 16354.736} C_VEL
LIN {X 0,Y 342.065,Z 307.575,A -85,B 0,C 180,E1 16352.871,E2 16352.871} C_VEL
LIN {X 0,Y 345.165,Z 313.605,A -85,B 0,C 180,E1 16350.498,E2 16350.498} C_VEL
LIN {X 0,Y 348.027,Z 319.264,A -85,B 0,C 180,E1 16348.474,E2 16348.474} C_VEL
LIN {X 0,Y 350.068,Z 322.346,A -85,B 0,C 180,E1 16347.571,E2 16347.571} C_VEL
LIN {X 0,Y 359.613,Z 335.297,A -85,B 0,C 180,E1 16344.56,E2 16344.56} C_VEL
LIN {X 0,Y 369.952,Z 350.8,A -85,B 0,C 180,E1 16341.664,E2 16341.664} C_VEL
LIN {X 0,Y 379.395,Z 365.951,A -85,B 0,C 180,E1 16339.287,E2 16339.287} C_VEL
LIN {X 0,Y 386.956,Z 379.474,A -85,B 0,C 180,E1 16337.516,E2 16337.516} C_VEL
LIN {X 0,Y 377.512,Z 596,A -85,B 0,C 180,E1 16333.402,E2 16333.402} C_VEL
LIN {X 0,Y 375.539,Z 617.023,A -85,B 0,C 180,E1 16332.765,E2 16332.765} C_VEL
LIN {X 0,Y 372.954,Z 636.489,A -85,B 0,C 180,E1 16331.928,E2 16331.928} C_VEL
LIN {X 0,Y 369.581,Z 656.478,A -85,B 0,C 180,E1 16330.793,E2 16330.793} C_VEL
LIN {X 0,Y 365.799,Z 675.03,A -85,B 0,C 180,E1 16329.456,E2 16329.456} C_VEL
LIN {X 0,Y 361.485,Z 693.207,A -85,B 0,C 180,E1 16327.818,E2 16327.818} C_VEL
LIN {X 0,Y 356.969,Z 710.053,A -85,B 0,C 180,E1 16325.954,E2 16325.954} C_VEL
LIN {X 0,Y 352.268,Z 726.154,A -85,B 0,C 180,E1 16323.8,E2 16323.8} C_VEL
LIN {X 0,Y 347.617,Z 741.168,A -85,B 0,C 180,E1 16321.373,E2 16321.373} C_VEL
LIN {X 0,Y 343.244,Z 754.755,A -85,B 0,C 180,E1 16318.726,E2 16318.726} C_VEL
LIN {X 0,Y 339.069,Z 767.528,A -85,B 0,C 180,E1 16315.688,E2 16315.688} C_VEL
LIN {X 0,Y 335.623,Z 778.284,A -85,B 0,C 180,E1 16312.552,E2 16312.552} C_VEL
LIN {X 0,Y 332.749,Z 787.841,A -85,B 0,C 180,E1 16309.118,E2 16309.118} C_VEL
LIN {X 0,Y 330.6,Z 795.918,A -85,B 0,C 180,E1 16305.435,E2 16305.435} C_VEL
LIN {X 0,Y 329.298,Z 801.822,A -85,B 0,C 180,E1 16301.915,E2 16301.915} C_VEL
LIN {X 0,Y 328.55,Z 806.288,A -85,B 0,C 180,E1 16298.223,E2 16298.223} C_VEL
LIN {X 0,Y 328.218,Z 809.016,A -85,B 0,C 180,E1 16294.543,E2 16294.543} C_VEL
LIN {X 0,Y 328.129,Z 810.147,A -85,B 0,C 180,E1 16291.048,E2 16291.048} C_VEL
LIN {X 0,Y 328.143,Z 809.918,A -85,B 0,C 180,E1 16287.555,E2 16287.555} C_VEL
LIN {X 0,Y 328.296,Z 808.234,A -85,B 0,C 180,E1 16284.057,E2 16284.057} C_VEL
LIN {X 0,Y 328.728,Z 805.057,A -85,B 0,C 180,E1 16280.547,E2 16280.547} C_VEL
LIN {X 0,Y 329.06,Z 803.087,A -85,B 0,C 180,E1 16278.916,E2 16278.916} C_VEL
LIN {X 0,Y 328.425,Z 801.41,A -85,B 0,C 180,E1 16277.6,E2 16277.6} C_VEL
LIN {X 0,Y 323.592,Z 796.361,A -85,B 0,C 180,E1 16274.066,E2 16274.066} C_VEL
LIN {X 0,Y 323.416,Z 794.216,A -85,B 0,C 180,E1 16272.946,E2 16272.946} C_VEL
LIN {X 0,Y 325.875,Z 785.938,A -85,B 0,C 180,E1 16269.339,E2 16269.339} C_VEL
LIN {X 0,Y 329.023,Z 776.184,A -85,B 0,C 180,E1 16265.971,E2 16265.971} C_VEL
LIN {X 0,Y 332.819,Z 765.021,A -85,B 0,C 180,E1 16262.83,E2 16262.83} C_VEL
LIN {X 0,Y 337.415,Z 751.644,A -85,B 0,C 180,E1 16259.752,E2 16259.752} C_VEL
LIN {X 0,Y 342.176,Z 737.498,A -85,B 0,C 180,E1 16257.079,E2 16257.079} C_VEL
LIN {X 0,Y 347.049,Z 722.395,A -85,B 0,C 180,E1 16254.716,E2 16254.716} C_VEL
LIN {X 0,Y 352.01,Z 705.63,A -85,B 0,C 180,E1 16252.567,E2 16252.567} C_VEL
LIN {X 0,Y 356.58,Z 688.62,A -85,B 0,C 180,E1 16250.781,E2 16250.781} C_VEL
LIN {X 0,Y 361.013,Z 669.988,A -85,B 0,C 180,E1 16249.186,E2 16249.186} C_VEL
LIN {X 0,Y 364.761,Z 651.57,A -85,B 0,C 180,E1 16247.918,E2 16247.918} C_VEL
LIN {X 0,Y 368.039,Z 631.798,A -85,B 0,C 180,E1 16246.861,E2 16246.861} C_VEL
LIN {X 0,Y 370.592,Z 611.459,A -85,B 0,C 180,E1 16246.061,E2 16246.061} C_VEL
LIN {X 0,Y 372.361,Z 590.291,A -85,B 0,C 180,E1 16245.491,E2 16245.491} C_VEL
LIN {X 0,Y 381.697,Z 382.702,A -85,B 0,C 180,E1 16241.509,E2 16241.509} C_VEL
LIN {X 0,Y 372.867,Z 367.294,A -85,B 0,C 180,E1 16239.335,E2 16239.335} C_VEL
LIN {X 0,Y 364.055,Z 353.134,A -85,B 0,C 180,E1 16236.976,E2 16236.976} C_VEL
LIN {X 0,Y 355.315,Z 340.202,A -85,B 0,C 180,E1 16234.397,E2 16234.397} C_VEL
LIN {X 0,Y 349.213,Z 331.84,A -85,B 0,C 180,E1 16232.421,E2 16232.421} C_VEL
LIN {X 0,Y 344.524,Z 325.523,A -85,B 0,C 180,E1 16230.769,E2 16230.769} C_VEL
LIN {X 0,Y 340.164,Z 319.479,A -85,B 0,C 180,E1 16229.012,E2 16229.012} C_VEL
LIN {X 0,Y 336.826,Z 313.313,A -85,B 0,C 180,E1 16226.441,E2 16226.441} C_VEL
LIN {X 0,Y 334.422,Z 308.794,A -85,B 0,C 180,E1 16224.368,E2 16224.368} C_VEL
LIN {X 0,Y 332.201,Z 304.753,A -85,B 0,C 180,E1 16222.287,E2 16222.287} C_VEL
LIN {X 0,Y 329.284,Z 299.943,A -85,B 0,C 180,E1 16219.328,E2 16219.328} C_VEL
LIN {X 0,Y 328.571,Z 298.57,A -85,B 0,C 180,E1 16218.45,E2 16218.45} C_VEL
LIN {X 0,Y 326.127,Z 294.946,A -85,B 0,C 180,E1 16215.47,E2 16215.47} C_VEL
LIN {X 0,Y 325.191,Z 293.022,A -85,B 0,C 180,E1 16213.877,E2 16213.877} C_VEL
LIN {X 0,Y 322.116,Z 287.914,A -85,B 0,C 180,E1 16206.416,E2 16206.416} C_VEL
LIN {X 0,Y 322.08,Z 287.656,A -85,B 0,C 180,E1 16201.957,E2 16201.957} C_VEL
LIN {X 0,Y 322.1,Z 287.763,A -85,B 0,C 180,E1 16197.688,E2 16197.688} C_VEL
LIN {X 0,Y 322.349,Z 288.911,A -85,B 0,C 180,E1 16195.018,E2 16195.018} C_VEL
LIN {X 0,Y 325.723,Z 293.681,A -85,B 0,C 180,E1 16188.67,E2 16188.67} C_VEL
LIN {X 0,Y 327.899,Z 297.868,A -85,B 0,C 180,E1 16185.52,E2 16185.52} C_VEL
LIN {X 0,Y 329.262,Z 299.59,A -85,B 0,C 180,E1 16184.14,E2 16184.14} C_VEL
LIN {X 0,Y 331.322,Z 303.429,A -85,B 0,C 180,E1 16181.891,E2 16181.891} C_VEL
LIN {X 0,Y 332.354,Z 304.709,A -85,B 0,C 180,E1 16181.04,E2 16181.04} C_VEL
LIN {X 0,Y 334.815,Z 309.125,A -85,B 0,C 180,E1 16178.818,E2 16178.818} C_VEL
LIN {X 0,Y 336.259,Z 311.794,A -85,B 0,C 180,E1 16177.721,E2 16177.721} C_VEL
LIN {X 0,Y 340.517,Z 316.838,A -85,B 0,C 180,E1 16175.958,E2 16175.958} C_VEL
LIN {X 0,Y 345.271,Z 322.724,A -85,B 0,C 180,E1 16174.162,E2 16174.162} C_VEL
LIN {X 0,Y 349.421,Z 327.998,A -85,B 0,C 180,E1 16172.707,E2 16172.707} C_VEL
LIN {X 0,Y 353.077,Z 332.725,A -85,B 0,C 180,E1 16171.5,E2 16171.5} C_VEL
LIN {X 0,Y 359.786,Z 341.758,A -85,B 0,C 180,E1 16169.432,E2 16169.432} C_VEL
LIN {X 0,Y 368.745,Z 354.884,A -85,B 0,C 180,E1 16166.908,E2 16166.908} C_VEL
LIN {X 0,Y 377.878,Z 369.283,A -85,B 0,C 180,E1 16164.564,E2 16164.564} C_VEL
LIN {X 0,Y 384.126,Z 380.159,A -85,B 0,C 180,E1 16163.058,E2 16163.058} C_VEL
LIN {X 0,Y 372.667,Z 596.512,A -85,B 0,C 180,E1 16158.616,E2 16158.616} C_VEL
LIN {X 0,Y 370.745,Z 618.583,A -85,B 0,C 180,E1 16158.026,E2 16158.026} C_VEL
LIN {X 0,Y 367.954,Z 639.704,A -85,B 0,C 180,E1 16157.223,E2 16157.223} C_VEL
LIN {X 0,Y 364.519,Z 660.452,A -85,B 0,C 180,E1 16156.168,E2 16156.168} C_VEL
LIN {X 0,Y 360.58,Z 680.548,A -85,B 0,C 180,E1 16154.872,E2 16154.872} C_VEL
LIN {X 0,Y 356.025,Z 700.674,A -85,B 0,C 180,E1 16153.254,E2 16153.254} C_VEL
LIN {X 0,Y 351.3,Z 719.305,A -85,B 0,C 180,E1 16151.41,E2 16151.41} C_VEL
LIN {X 0,Y 346.207,Z 738.078,A -85,B 0,C 180,E1 16149.165,E2 16149.165} C_VEL
LIN {X 0,Y 341.466,Z 754.608,A -85,B 0,C 180,E1 16146.809,E2 16146.809} C_VEL
LIN {X 0,Y 336.741,Z 770.652,A -85,B 0,C 180,E1 16144.065,E2 16144.065} C_VEL
LIN {X 0,Y 332.499,Z 784.983,A -85,B 0,C 180,E1 16141.145,E2 16141.145} C_VEL
LIN {X 0,Y 328.719,Z 798.286,A -85,B 0,C 180,E1 16137.931,E2 16137.931} C_VEL
LIN {X 0,Y 325.586,Z 810.206,A -85,B 0,C 180,E1 16134.492,E2 16134.492} C_VEL
LIN {X 0,Y 323.164,Z 820.55,A -85,B 0,C 180,E1 16130.842,E2 16130.842} C_VEL
LIN {X 0,Y 321.539,Z 829.009,A -85,B 0,C 180,E1 16127.182,E2 16127.182} C_VEL
LIN {X 0,Y 320.586,Z 835.773,A -85,B 0,C 180,E1 16123.527,E2 16123.527} C_VEL
LIN {X 0,Y 320.151,Z 840.782,A -85,B 0,C 180,E1 16119.89,E2 16119.89} C_VEL
LIN {X 0,Y 320.033,Z 844.253,A -85,B 0,C 180,E1 16116.278,E2 16116.278} C_VEL
LIN {X 0,Y 320.053,Z 846.039,A -85,B 0,C 180,E1 16113.044,E2 16113.044} C_VEL
LIN {X 0,Y 320.065,Z 846.586,A -85,B 0,C 180,E1 16109.463,E2 16109.463} C_VEL
LIN {X 0,Y 320.044,Z 845.74,A -85,B 0,C 180,E1 16106.238,E2 16106.238} C_VEL
LIN {X 0,Y 320.053,Z 843.377,A -85,B 0,C 180,E1 16102.641,E2 16102.641} C_VEL
LIN {X 0,Y 320.227,Z 839.665,A -85,B 0,C 180,E1 16099.203,E2 16099.203} C_VEL
LIN {X 0,Y 320.812,Z 833.875,A -85,B 0,C 180,E1 16095.378,E2 16095.378} C_VEL
LIN {X 0,Y 321.953,Z 826.7,A -85,B 0,C 180,E1 16091.72,E2 16091.72} C_VEL
LIN {X 0,Y 323.804,Z 817.622,A -85,B 0,C 180,E1 16088.061,E2 16088.061} C_VEL
LIN {X 0,Y 326.322,Z 807.182,A -85,B 0,C 180,E1 16084.599,E2 16084.599} C_VEL
LIN {X 0,Y 329.687,Z 794.789,A -85,B 0,C 180,E1 16081.171,E2 16081.171} C_VEL
LIN {X 0,Y 333.703,Z 780.931,A -85,B 0,C 180,E1 16077.973,E2 16077.973} C_VEL
LIN {X 0,Y 338.089,Z 765.946,A -85,B 0,C 180,E1 16075.094,E2 16075.094} C_VEL
LIN {X 0,Y 342.882,Z 749.609,A -85,B 0,C 180,E1 16072.451,E2 16072.451} C_VEL
LIN {X 0,Y 347.749,Z 732.478,A -85,B 0,C 180,E1 16070.122,E2 16070.122} C_VEL
LIN {X 0,Y 352.726,Z 713.797,A -85,B 0,C 180,E1 16068.013,E2 16068.013} C_VEL
LIN {X 0,Y 357.293,Z 695.054,A -85,B 0,C 180,E1 16066.275,E2 16066.275} C_VEL
LIN {X 0,Y 361.725,Z 674.766,A -85,B 0,C 180,E1 16064.735,E2 16064.735} C_VEL
LIN {X 0,Y 365.609,Z 654.15,A -85,B 0,C 180,E1 16063.481,E2 16063.481} C_VEL
LIN {X 0,Y 368.932,Z 632.407,A -85,B 0,C 180,E1 16062.476,E2 16062.476} C_VEL
LIN {X 0,Y 371.495,Z 610.555,A -85,B 0,C 180,E1 16061.747,E2 16061.747} C_VEL
LIN {X 0,Y 373.393,Z 582.232,A -85,B 0,C 180,E1 16061.086,E2 16061.086} C_VEL
LIN {X 0,Y 384.049,Z 379.8,A -85,B 0,C 180,E1 16056.939,E2 16056.939} C_VEL
LIN {X 0,Y 373.263,Z 361.802,A -85,B 0,C 180,E1 16054.3,E2 16054.3} C_VEL
LIN {X 0,Y 363.419,Z 346.99,A -85,B 0,C 180,E1 16051.655,E2 16051.655} C_VEL
LIN {X 0,Y 354.797,Z 334.966,A -85,B 0,C 180,E1 16049.086,E2 16049.086} C_VEL
LIN {X 0,Y 349.639,Z 328.299,A -85,B 0,C 180,E1 16047.413,E2 16047.413} C_VEL
LIN {X 0,Y 345.57,Z 323.113,A -85,B 0,C 180,E1 16045.998,E2 16045.998} C_VEL
LIN {X 0,Y 340.88,Z 317.315,A -85,B 0,C 180,E1 16044.245,E2 16044.245} C_VEL
LIN {X 0,Y 338.151,Z 314.063,A -85,B 0,C 180,E1 16043.157,E2 16043.157} C_VEL
LIN {X 0,Y 335.74,Z 310.913,A -85,B 0,C 180,E1 16042.039,E2 16042.039} C_VEL
LIN {X 0,Y 334.71,Z 309.013,A -85,B 0,C 180,E1 16041.189,E2 16041.189} C_VEL
LIN {X 0,Y 332.285,Z 304.51,A -85,B 0,C 180,E1 16038.964,E2 16038.964} C_VEL
LIN {X 0,Y 329.664,Z 300.752,A -85,B 0,C 180,E1 16036.564,E2 16036.564} C_VEL
LIN {X 0,Y 328.678,Z 298.677,A -85,B 0,C 180,E1 16035.346,E2 16035.346} C_VEL
LIN {X 0,Y 326.167,Z 295.003,A -85,B 0,C 180,E1 16032.391,E2 16032.391} C_VEL
LIN {X 0,Y 325.192,Z 293.062,A -85,B 0,C 180,E1 16030.81,E2 16030.81} C_VEL
LIN {X 0,Y 322.091,Z 287.867,A -85,B 0,C 180,E1 16023.559,E2 16023.559} C_VEL
LIN {X 0,Y 322.065,Z 287.626,A -85,B 0,C 180,E1 16019.288,E2 16019.288} C_VEL
LIN {X 0,Y 322.099,Z 287.679,A -85,B 0,C 180,E1 16014.835,E2 16014.835} C_VEL
LIN {X 0,Y 322.199,Z 288.213,A -85,B 0,C 180,E1 16012.331,E2 16012.331} C_VEL
LIN {X 0,Y 325.742,Z 293.805,A -85,B 0,C 180,E1 16005.058,E2 16005.058} C_VEL
LIN {X 0,Y 327.816,Z 297.793,A -85,B 0,C 180,E1 16002.058,E2 16002.058} C_VEL
LIN {X 0,Y 329.048,Z 299.214,A -85,B 0,C 180,E1 16000.842,E2 16000.842} C_VEL
LIN {X 0,Y 330.827,Z 302.873,A -85,B 0,C 180,E1 15998.735,E2 15998.735} C_VEL
LIN {X 0,Y 332.211,Z 304.805,A -85,B 0,C 180,E1 15997.511,E2 15997.511} C_VEL
LIN {X 0,Y 334.442,Z 308.822,A -85,B 0,C 180,E1 15995.445,E2 15995.445} C_VEL
LIN {X 0,Y 337.797,Z 315.126,A -85,B 0,C 180,E1 15992.618,E2 15992.618} C_VEL
LIN {X 0,Y 340.437,Z 320.086,A -85,B 0,C 180,E1 15990.654,E2 15990.654} C_VEL
LIN {X 0,Y 347.809,Z 329.925,A -85,B 0,C 180,E1 15987.919,E2 15987.919} C_VEL
LIN {X 0,Y 354.644,Z 339.318,A -85,B 0,C 180,E1 15985.676,E2 15985.676} C_VEL
LIN {X 0,Y 363.356,Z 352.167,A -85,B 0,C 180,E1 15983.089,E2 15983.089} C_VEL
LIN {X 0,Y 372.48,Z 366.689,A -85,B 0,C 180,E1 15980.639,E2 15980.639} C_VEL
LIN {X 0,Y 381.519,Z 382.467,A -85,B 0,C 180,E1 15978.417,E2 15978.417} C_VEL
LIN {X 0,Y 381.612,Z 384.557,A -85,B 0,C 180,E1 15978.341,E2 15978.341} C_VEL
LIN {X 0,Y 371.94,Z 596.26,A -85,B 0,C 180,E1 15974.28,E2 15974.28} C_VEL
LIN {X 0,Y 369.868,Z 617.477,A -85,B 0,C 180,E1 15973.631,E2 15973.631} C_VEL
LIN {X 0,Y 367.089,Z 637.519,A -85,B 0,C 180,E1 15972.756,E2 15972.756} C_VEL
LIN {X 0,Y 363.571,Z 657.422,A -85,B 0,C 180,E1 15971.605,E2 15971.605} C_VEL
LIN {X 0,Y 359.673,Z 675.741,A -85,B 0,C 180,E1 15970.264,E2 15970.264} C_VEL
LIN {X 0,Y 355.2,Z 693.867,A -85,B 0,C 180,E1 15968.61,E2 15968.61} C_VEL
LIN {X 0,Y 350.465,Z 710.791,A -85,B 0,C 180,E1 15966.709,E2 15966.709} C_VEL
LIN {X 0,Y 345.609,Z 726.715,A -85,B 0,C 180,E1 15964.543,E2 15964.543} C_VEL
LIN {X 0,Y 340.749,Z 741.696,A -85,B 0,C 180,E1 15962.079,E2 15962.079} C_VEL
LIN {X 0,Y 336.118,Z 755.412,A -85,B 0,C 180,E1 15959.355,E2 15959.355} C_VEL
LIN {X 0,Y 331.788,Z 768.027,A -85,B 0,C 180,E1 15956.294,E2 15956.294} C_VEL
LIN {X 0,Y 328.194,Z 778.627,A -85,B 0,C 180,E1 15953.141,E2 15953.141} C_VEL
LIN {X 0,Y 325.235,Z 787.878,A -85,B 0,C 180,E1 15949.765,E2 15949.765} C_VEL
LIN {X 0,Y 322.991,Z 795.715,A -85,B 0,C 180,E1 15946.177,E2 15946.177} C_VEL
LIN {X 0,Y 321.517,Z 801.804,A -85,B 0,C 180,E1 15942.573,E2 15942.573} C_VEL
LIN {X 0,Y 320.654,Z 806.366,A -85,B 0,C 180,E1 15938.788,E2 15938.788} C_VEL
LIN {X 0,Y 320.27,Z 809.151,A -85,B 0,C 180,E1 15935.19,E2 15935.19} C_VEL
LIN {X 0,Y 320.14,Z 810.554,A -85,B 0,C 180,E1 15931.432,E2 15931.432} C_VEL
LIN {X 0,Y 320.153,Z 810.483,A -85,B 0,C 180,E1 15927.852,E2 15927.852} C_VEL
LIN {X 0,Y 320.296,Z 808.895,A -85,B 0,C 180,E1 15924.267,E2 15924.267} C_VEL
LIN {X 0,Y 320.76,Z 805.704,A -85,B 0,C 180,E1 15920.491,E2 15920.491} C_VEL
LIN {X 0,Y 321.663,Z 801.127,A -85,B 0,C 180,E1 15916.885,E2 15916.885} C_VEL
LIN {X 0,Y 323.333,Z 794.548,A -85,B 0,C 180,E1 15913.102,E2 15913.102} C_VEL
LIN {X 0,Y 323.416,Z 794.216,A -85,B 0,C 180,E1 15912.946,E2 15912.946} C_VEL
LIN {X 0,Y 323.185,Z 791.641,A -85,B 0,C 180,E1 15911.653,E2 15911.653} C_VEL
LIN {X 0,Y 319.706,Z 784.882,A -85,B 0,C 180,E1 15908.328,E2 15908.328} C_VEL
LIN {X 0,Y 319.901,Z 781.658,A -85,B 0,C 180,E1 15907.055,E2 15907.055} C_VEL
LIN {X 0,Y 323.525,Z 771.337,A -85,B 0,C 180,E1 15903.773,E2 15903.773} C_VEL
LIN {X 0,Y 327.936,Z 759.137,A -85,B 0,C 180,E1 15900.602,E2 15900.602} C_VEL
LIN {X 0,Y 332.553,Z 746.287,A -85,B 0,C 180,E1 15897.849,E2 15897.849} C_VEL
LIN {X 0,Y 337.586,Z 731.8,A -85,B 0,C 180,E1 15895.278,E2 15895.278} C_VEL
LIN {X 0,Y 342.749,Z 715.838,A -85,B 0,C 180,E1 15892.96,E2 15892.96} C_VEL
LIN {X 0,Y 347.706,Z 699.182,A -85,B 0,C 180,E1 15890.969,E2 15890.969} C_VEL
LIN {X 0,Y 352.569,Z 680.9,A -85,B 0,C 180,E1 15889.182,E2 15889.182} C_VEL
LIN {X 0,Y 356.826,Z 662.639,A -85,B 0,C 180,E1 15887.741,E2 15887.741} C_VEL
LIN {X 0,Y 360.684,Z 642.782,A -85,B 0,C 180,E1 15886.507,E2 15886.507} C_VEL
LIN {X 0,Y 363.7,Z 622.998,A -85,B 0,C 180,E1 15885.579,E2 15885.579} C_VEL
LIN {X 0,Y 366.014,Z 602.17,A -85,B 0,C 180,E1 15884.871,E2 15884.871} C_VEL
LIN {X 0,Y 367.609,Z 576.785,A -85,B 0,C 180,E1 15884.307,E2 15884.307} C_VEL
LIN {X 0,Y 376.541,Z 386.244,A -85,B 0,C 180,E1 15880.635,E2 15880.635} C_VEL
LIN {X 0,Y 367.593,Z 370.589,A -85,B 0,C 180,E1 15878.328,E2 15878.328} C_VEL
LIN {X 0,Y 358.313,Z 355.765,A -85,B 0,C 180,E1 15875.708,E2 15875.708} C_VEL
LIN {X 0,Y 350.382,Z 344.04,A -85,B 0,C 180,E1 15873.223,E2 15873.223} C_VEL
LIN {X 0,Y 342.744,Z 333.494,A -85,B 0,C 180,E1 15870.553,E2 15870.553} C_VEL
LIN {X 0,Y 336.199,Z 324.885,A -85,B 0,C 180,E1 15867.972,E2 15867.972} C_VEL
LIN {X 0,Y 331.886,Z 319.312,A -85,B 0,C 180,E1 15866.03,E2 15866.03} C_VEL
LIN {X 0,Y 329.725,Z 315.152,A -85,B 0,C 180,E1 15864.115,E2 15864.115} C_VEL
LIN {X 0,Y 327.081,Z 310.279,A -85,B 0,C 180,E1 15861.521,E2 15861.521} C_VEL
LIN {X 0,Y 324.809,Z 306.445,A -85,B 0,C 180,E1 15859.089,E2 15859.089} C_VEL
LIN {X 0,Y 323.998,Z 305.025,A -85,B 0,C 180,E1 15858.11,E2 15858.11} C_VEL
LIN {X 0,Y 321.752,Z 301.387,A -85,B 0,C 180,E1 15855.132,E2 15855.132} C_VEL
LIN {X 0,Y 320.919,Z 299.747,A -85,B 0,C 180,E1 15853.697,E2 15853.697} C_VEL
LIN {X 0,Y 317.881,Z 294.685,A -85,B 0,C 180,E1 15846.321,E2 15846.321} C_VEL
LIN {X 0,Y 317.226,Z 293.991,A -85,B 0,C 180,E1 15841.265,E2 15841.265} C_VEL
LIN {X 0,Y 317.966,Z 294.854,A -85,B 0,C 180,E1 15836.575,E2 15836.575} C_VEL
LIN {X 0,Y 321.563,Z 300.643,A -85,B 0,C 180,E1 15828.704,E2 15828.704} C_VEL
LIN {X 0,Y 323.784,Z 304.746,A -85,B 0,C 180,E1 15825.515,E2 15825.515} C_VEL
LIN {X 0,Y 324.937,Z 306.317,A -85,B 0,C 180,E1 15824.289,E2 15824.289} C_VEL
LIN {X 0,Y 326.994,Z 310.121,A -85,B 0,C 180,E1 15822.012,E2 15822.012} C_VEL
LIN {X 0,Y 328.066,Z 311.736,A -85,B 0,C 180,E1 15821.06,E2 15821.06} C_VEL
LIN {X 0,Y 331.995,Z 316.443,A -85,B 0,C 180,E1 15819.092,E2 15819.092} C_VEL
LIN {X 0,Y 338.339,Z 324.205,A -85,B 0,C 180,E1 15816.349,E2 15816.349} C_VEL
LIN {X 0,Y 345.527,Z 333.186,A -85,B 0,C 180,E1 15813.629,E2 15813.629} C_VEL
LIN {X 0,Y 353.415,Z 343.789,A -85,B 0,C 180,E1 15810.975,E2 15810.975} C_VEL
LIN {X 0,Y 362.945,Z 357.56,A -85,B 0,C 180,E1 15808.114,E2 15808.114} C_VEL
LIN {X 0,Y 373.284,Z 373.9,A -85,B 0,C 180,E1 15805.33,E2 15805.33} C_VEL
LIN {X 0,Y 378.882,Z 383.793,A -85,B 0,C 180,E1 15803.92,E2 15803.92} C_VEL
LIN {X 0,Y 367.11,Z 597.51,A -85,B 0,C 180,E1 15799.497,E2 15799.497} C_VEL
LIN {X 0,Y 365.055,Z 619.603,A -85,B 0,C 180,E1 15798.891,E2 15798.891} C_VEL
LIN {X 0,Y 362.172,Z 640.592,A -85,B 0,C 180,E1 15798.08,E2 15798.08} C_VEL
LIN {X 0,Y 358.664,Z 660.819,A -85,B 0,C 180,E1 15797.034,E2 15797.034} C_VEL
LIN {X 0,Y 354.374,Z 681.689,A -85,B 0,C 180,E1 15795.662,E2 15795.662} C_VEL
LIN {X 0,Y 349.862,Z 700.856,A -85,B 0,C 180,E1 15794.097,E2 15794.097} C_VEL
LIN {X 0,Y 344.859,Z 719.72,A -85,B 0,C 180,E1 15792.2,E2 15792.2} C_VEL
LIN {X 0,Y 339.566,Z 738.334,A -85,B 0,C 180,E1 15789.933,E2 15789.933} C_VEL
LIN {X 0,Y 334.557,Z 754.956,A -85,B 0,C 180,E1 15787.511,E2 15787.511} C_VEL
LIN {X 0,Y 329.596,Z 771.021,A -85,B 0,C 180,E1 15784.705,E2 15784.705} C_VEL
LIN {X 0,Y 325.146,Z 785.254,A -85,B 0,C 180,E1 15781.724,E2 15781.724} C_VEL
LIN {X 0,Y 320.982,Z 799.104,A -85,B 0,C 180,E1 15778.26,E2 15778.26} C_VEL
LIN {X 0,Y 317.732,Z 810.799,A -85,B 0,C 180,E1 15774.741,E2 15774.741} C_VEL
LIN {X 0,Y 315.228,Z 821.028,A -85,B 0,C 180,E1 15771.003,E2 15771.003} C_VEL
LIN {X 0,Y 313.55,Z 829.282,A -85,B 0,C 180,E1 15767.251,E2 15767.251} C_VEL
LIN {X 0,Y 312.545,Z 836.123,A -85,B 0,C 180,E1 15763.316,E2 15763.316} C_VEL
LIN {X 0,Y 312.135,Z 840.985,A -85,B 0,C 180,E1 15759.588,E2 15759.588} C_VEL
LIN {X 0,Y 312.042,Z 844.047,A -85,B 0,C 180,E1 15756.07,E2 15756.07} C_VEL
LIN {X 0,Y 312.065,Z 845.808,A -85,B 0,C 180,E1 15752.571,E2 15752.571} C_VEL
LIN {X 0,Y 312.081,Z 846.09,A -85,B 0,C 180,E1 15749.082,E2 15749.082} C_VEL
LIN {X 0,Y 312.05,Z 845.142,A -85,B 0,C 180,E1 15745.774,E2 15745.774} C_VEL
LIN {X 0,Y 312.069,Z 842.577,A -85,B 0,C 180,E1 15742.081,E2 15742.081} C_VEL
LIN {X 0,Y 312.306,Z 838.535,A -85,B 0,C 180,E1 15738.364,E2 15738.364} C_VEL
LIN {X 0,Y 312.985,Z 832.756,A -85,B 0,C 180,E1 15734.625,E2 15734.625} C_VEL
LIN {X 0,Y 314.375,Z 824.927,A -85,B 0,C 180,E1 15730.685,E2 15730.685} C_VEL
LIN {X 0,Y 316.496,Z 815.649,A -85,B 0,C 180,E1 15726.938,E2 15726.938} C_VEL
LIN {X 0,Y 319.334,Z 804.869,A -85,B 0,C 180,E1 15723.402,E2 15723.402} C_VEL
LIN {X 0,Y 322.832,Z 792.8,A -85,B 0,C 180,E1 15720.091,E2 15720.091} C_VEL
LIN {X 0,Y 327.12,Z 778.841,A -85,B 0,C 180,E1 15716.876,E2 15716.876} C_VEL
LIN {X 0,Y 331.923,Z 763.47,A -85,B 0,C 180,E1 15713.922,E2 15713.922} C_VEL
LIN {X 0,Y 336.892,Z 747.155,A -85,B 0,C 180,E1 15711.311,E2 15711.311} C_VEL
LIN {X 0,Y 342.198,Z 729.097,A -85,B 0,C 180,E1 15708.898,E2 15708.898} C_VEL
LIN {X 0,Y 347.177,Z 711.125,A -85,B 0,C 180,E1 15706.9,E2 15706.9} C_VEL
LIN {X 0,Y 351.959,Z 692.017,A -85,B 0,C 180,E1 15705.153,E2 15705.153} C_VEL
LIN {X 0,Y 356.233,Z 672.757,A -85,B 0,C 180,E1 15703.721,E2 15703.721} C_VEL
LIN {X 0,Y 360.236,Z 651.846,A -85,B 0,C 180,E1 15702.474,E2 15702.474} C_VEL
LIN {X 0,Y 363.662,Z 630.113,A -85,B 0,C 180,E1 15701.486,E2 15701.486} C_VEL
LIN {X 0,Y 366.217,Z 608.063,A -85,B 0,C 180,E1 15700.775,E2 15700.775} C_VEL
LIN {X 0,Y 368.239,Z 576.415,A -85,B 0,C 180,E1 15700.057,E2 15700.057} C_VEL
LIN {X 0,Y 378.813,Z 383.523,A -85,B 0,C 180,E1 15696.082,E2 15696.082} C_VEL
LIN {X 0,Y 369.185,Z 367.302,A -85,B 0,C 180,E1 15693.631,E2 15693.631} C_VEL
LIN {X 0,Y 359.964,Z 353.18,A -85,B 0,C 180,E1 15691.061,E2 15691.061} C_VEL
LIN {X 0,Y 351.731,Z 341.542,A -85,B 0,C 180,E1 15688.526,E2 15688.526} C_VEL
LIN {X 0,Y 344.469,Z 331.835,A -85,B 0,C 180,E1 15686.041,E2 15686.041} C_VEL
LIN {X 0,Y 336.591,Z 321.976,A -85,B 0,C 180,E1 15682.993,E2 15682.993} C_VEL
LIN {X 0,Y 331.666,Z 316.16,A -85,B 0,C 180,E1 15680.838,E2 15680.838} C_VEL
LIN {X 0,Y 328.083,Z 311.758,A -85,B 0,C 180,E1 15679.031,E2 15679.031} C_VEL
LIN {X 0,Y 327.097,Z 310.222,A -85,B 0,C 180,E1 15678.167,E2 15678.167} C_VEL
LIN {X 0,Y 324.975,Z 306.444,A -85,B 0,C 180,E1 15675.892,E2 15675.892} C_VEL
LIN {X 0,Y 323.656,Z 304.612,A -85,B 0,C 180,E1 15674.491,E2 15674.491} C_VEL
LIN {X 0,Y 321.558,Z 300.669,A -85,B 0,C 180,E1 15671.478,E2 15671.478} C_VEL
LIN {X 0,Y 317.844,Z 294.619,A -85,B 0,C 180,E1 15663.426,E2 15663.426} C_VEL
LIN {X 0,Y 317.037,Z 293.827,A -85,B 0,C 180,E1 15658.192,E2 15658.192} C_VEL
LIN {X 0,Y 317.866,Z 294.635,A -85,B 0,C 180,E1 15653.135,E2 15653.135} C_VEL
LIN {X 0,Y 321.463,Z 300.513,A -85,B 0,C 180,E1 15645.223,E2 15645.223} C_VEL
LIN {X 0,Y 323.505,Z 304.507,A -85,B 0,C 180,E1 15642.159,E2 15642.159} C_VEL
LIN {X 0,Y 324.651,Z 305.991,A -85,B 0,C 180,E1 15640.946,E2 15640.946} C_VEL
LIN {X 0,Y 326.658,Z 309.809,A -85,B 0,C 180,E1 15638.639,E2 15638.639} C_VEL
LIN {X 0,Y 327.61,Z 311.203,A -85,B 0,C 180,E1 15637.762,E2 15637.762} C_VEL
LIN {X 0,Y 329.805,Z 315.254,A -85,B 0,C 180,E1 15635.65,E2 15635.65} C_VEL
LIN {X 0,Y 332.519,Z 320.066,A -85,B 0,C 180,E1 15633.478,E2 15633.478} C_VEL
LIN {X 0,Y 338.696,Z 328.164,A -85,B 0,C 180,E1 15630.85,E2 15630.85} C_VEL
LIN {X 0,Y 345.146,Z 336.836,A -85,B 0,C 180,E1 15628.424,E2 15628.424} C_VEL
LIN {X 0,Y 351.862,Z 346.234,A -85,B 0,C 180,E1 15626.154,E2 15626.154} C_VEL
LIN {X 0,Y 360.684,Z 359.495,A -85,B 0,C 180,E1 15623.465,E2 15623.465} C_VEL
LIN {X 0,Y 369.886,Z 374.561,A -85,B 0,C 180,E1 15620.937,E2 15620.937} C_VEL
LIN {X 0,Y 376.509,Z 386.421,A -85,B 0,C 180,E1 15619.251,E2 15619.251} C_VEL
LIN {X 0,Y 366.472,Z 596.314,A -85,B 0,C 180,E1 15615.189,E2 15615.189} C_VEL
LIN {X 0,Y 364.327,Z 617.525,A -85,B 0,C 180,E1 15614.538,E2 15614.538} C_VEL
LIN {X 0,Y 361.535,Z 637.068,A -85,B 0,C 180,E1 15613.685,E2 15613.685} C_VEL
LIN {X 0,Y 357.914,Z 657.018,A -85,B 0,C 180,E1 15612.534,E2 15612.534} C_VEL
LIN {X 0,Y 353.847,Z 675.561,A -85,B 0,C 180,E1 15611.175,E2 15611.175} C_VEL
LIN {X 0,Y 349.111,Z 694.038,A -85,B 0,C 180,E1 15609.479,E2 15609.479} C_VEL
LIN {X 0,Y 344.246,Z 710.773,A -85,B 0,C 180,E1 15607.584,E2 15607.584} C_VEL
LIN {X 0,Y 339.01,Z 727.273,A -85,B 0,C 180,E1 15605.314,E2 15605.314} C_VEL
LIN {X 0,Y 333.935,Z 742.222,A -85,B 0,C 180,E1 15602.815,E2 15602.815} C_VEL
LIN {X 0,Y 329.151,Z 755.766,A -85,B 0,C 180,E1 15600.08,E2 15600.08} C_VEL
LIN {X 0,Y 324.544,Z 768.525,A -85,B 0,C 180,E1 15596.928,E2 15596.928} C_VEL
LIN {X 0,Y 320.751,Z 779.11,A -85,B 0,C 180,E1 15593.71,E2 15593.71} C_VEL
LIN {X 0,Y 317.619,Z 788.35,A -85,B 0,C 180,E1 15590.259,E2 15590.259} C_VEL
LIN {X 0,Y 315.226,Z 796.179,A -85,B 0,C 180,E1 15586.586,E2 15586.586} C_VEL
LIN {X 0,Y 313.642,Z 802.262,A -85,B 0,C 180,E1 15582.894,E2 15582.894} C_VEL
LIN {X 0,Y 312.714,Z 806.821,A -85,B 0,C 180,E1 15579.013,E2 15579.013} C_VEL
LIN {X 0,Y 312.291,Z 809.616,A -85,B 0,C 180,E1 15575.297,E2 15575.297} C_VEL
LIN {X 0,Y 312.153,Z 811.002,A -85,B 0,C 180,E1 15571.468,E2 15571.468} C_VEL
LIN {X 0,Y 312.167,Z 810.931,A -85,B 0,C 180,E1 15567.797,E2 15567.797} C_VEL
LIN {X 0,Y 312.323,Z 809.345,A -85,B 0,C 180,E1 15564.12,E2 15564.12} C_VEL
LIN {X 0,Y 312.827,Z 806.158,A -85,B 0,C 180,E1 15560.247,E2 15560.247} C_VEL
LIN {X 0,Y 313.804,Z 801.586,A -85,B 0,C 180,E1 15556.55,E2 15556.55} C_VEL
LIN {X 0,Y 315.591,Z 795.014,A -85,B 0,C 180,E1 15552.674,E2 15552.674} C_VEL
LIN {X 0,Y 318.189,Z 786.714,A -85,B 0,C 180,E1 15548.952,E2 15548.952} C_VEL
LIN {X 0,Y 319.901,Z 781.658,A -85,B 0,C 180,E1 15547.055,E2 15547.055} C_VEL
LIN {X 0,Y 320.2,Z 778.34,A -85,B 0,C 180,E1 15545.799,E2 15545.799} C_VEL
LIN {X 0,Y 318.006,Z 769.067,A -85,B 0,C 180,E1 15542.393,E2 15542.393} C_VEL
LIN {X 0,Y 318.66,Z 765.546,A -85,B 0,C 180,E1 15541.378,E2 15541.378} C_VEL
LIN {X 0,Y 323.541,Z 752.661,A -85,B 0,C 180,E1 15538.308,E2 15538.308} C_VEL
LIN {X 0,Y 328.755,Z 738.565,A -85,B 0,C 180,E1 15535.551,E2 15535.551} C_VEL
LIN {X 0,Y 334.041,Z 723.513,A -85,B 0,C 180,E1 15533.121,E2 15533.121} C_VEL
LIN {X 0,Y 339.41,Z 706.81,A -85,B 0,C 180,E1 15530.92,E2 15530.92} C_VEL
LIN {X 0,Y 344.335,Z 689.924,A -85,B 0,C 180,E1 15529.097,E2 15529.097} C_VEL
LIN {X 0,Y 349.098,Z 671.478,A -85,B 0,C 180,E1 15527.475,E2 15527.475} C_VEL
LIN {X 0,Y 353.118,Z 653.342,A -85,B 0,C 180,E1 15526.189,E2 15526.189} C_VEL
LIN {X 0,Y 356.703,Z 633.3,A -85,B 0,C 180,E1 15525.092,E2 15525.092} C_VEL
LIN {X 0,Y 359.496,Z 612.978,A -85,B 0,C 180,E1 15524.267,E2 15524.267} C_VEL
LIN {X 0,Y 361.509,Z 591.156,A -85,B 0,C 180,E1 15523.66,E2 15523.66} C_VEL
LIN {X 0,Y 371.467,Z 389.892,A -85,B 0,C 180,E1 15519.738,E2 15519.738} C_VEL
LIN {X 0,Y 363.347,Z 375.585,A -85,B 0,C 180,E1 15517.555,E2 15517.555} C_VEL
LIN {X 0,Y 354.565,Z 361.329,A -85,B 0,C 180,E1 15514.971,E2 15514.971} C_VEL
LIN {X 0,Y 347.105,Z 350.178,A -85,B 0,C 180,E1 15512.544,E2 15512.544} C_VEL
LIN {X 0,Y 339.856,Z 339.996,A -85,B 0,C 180,E1 15509.912,E2 15509.912} C_VEL
LIN {X 0,Y 333.956,Z 332.071,A -85,B 0,C 180,E1 15507.505,E2 15507.505} C_VEL
LIN {X 0,Y 329.579,Z 326.428,A -85,B 0,C 180,E1 15505.518,E2 15505.518} C_VEL
LIN {X 0,Y 325.777,Z 321.734,A -85,B 0,C 180,E1 15503.611,E2 15503.611} C_VEL
LIN {X 0,Y 323.172,Z 318.006,A -85,B 0,C 180,E1 15501.985,E2 15501.985} C_VEL
LIN {X 0,Y 321.904,Z 316.025,A -85,B 0,C 180,E1 15500.738,E2 15500.738} C_VEL
LIN {X 0,Y 319.802,Z 311.858,A -85,B 0,C 180,E1 15498.116,E2 15498.116} C_VEL
LIN {X 0,Y 317.466,Z 308.099,A -85,B 0,C 180,E1 15494.967,E2 15494.967} C_VEL
LIN {X 0,Y 316.652,Z 306.475,A -85,B 0,C 180,E1 15493.513,E2 15493.513} C_VEL
LIN {X 0,Y 313.789,Z 301.538,A -85,B 0,C 180,E1 15486.212,E2 15486.212} C_VEL
LIN {X 0,Y 313.194,Z 300.912,A -85,B 0,C 180,E1 15481.098,E2 15481.098} C_VEL
LIN {X 0,Y 313.893,Z 301.705,A -85,B 0,C 180,E1 15476.713,E2 15476.713} C_VEL
LIN {X 0,Y 317.328,Z 307.326,A -85,B 0,C 180,E1 15468.919,E2 15468.919} C_VEL
LIN {X 0,Y 319.491,Z 311.447,A -85,B 0,C 180,E1 15465.686,E2 15465.686} C_VEL
LIN {X 0,Y 320.76,Z 312.996,A -85,B 0,C 180,E1 15464.543,E2 15464.543} C_VEL
LIN {X 0,Y 324.118,Z 317.234,A -85,B 0,C 180,E1 15462.496,E2 15462.496} C_VEL
LIN {X 0,Y 326.08,Z 319.19,A -85,B 0,C 180,E1 15461.451,E2 15461.451} C_VEL
LIN {X 0,Y 330.306,Z 324.125,A -85,B 0,C 180,E1 15459.351,E2 15459.351} C_VEL
LIN {X 0,Y 337.035,Z 332.678,A -85,B 0,C 180,E1 15456.391,E2 15456.391} C_VEL
LIN {X 0,Y 343.656,Z 341.262,A -85,B 0,C 180,E1 15453.846,E2 15453.846} C_VEL
LIN {X 0,Y 350.36,Z 350.325,A -85,B 0,C 180,E1 15451.538,E2 15451.538} C_VEL
LIN {X 0,Y 359.718,Z 364.099,A -85,B 0,C 180,E1 15448.636,E2 15448.636} C_VEL
LIN {X 0,Y 369.636,Z 380.084,A -85,B 0,C 180,E1 15445.879,E2 15445.879} C_VEL
LIN {X 0,Y 373.722,Z 387.499,A -85,B 0,C 180,E1 15444.805,E2 15444.805} C_VEL
LIN {X 0,Y 361.658,Z 598.312,A -85,B 0,C 180,E1 15440.41,E2 15440.41} C_VEL
LIN {X 0,Y 359.43,Z 620.801,A -85,B 0,C 180,E1 15439.776,E2 15439.776} C_VEL
LIN {X 0,Y 356.378,Z 642.111,A -85,B 0,C 180,E1 15438.937,E2 15438.937} C_VEL
LIN {X 0,Y 352.575,Z 662.86,A -85,B 0,C 180,E1 15437.83,E2 15437.83} C_VEL
LIN {X 0,Y 348.013,Z 683.775,A -85,B 0,C 180,E1 15436.407,E2 15436.407} C_VEL
LIN {X 0,Y 343.086,Z 703.526,A -85,B 0,C 180,E1 15434.731,E2 15434.731} C_VEL
LIN {X 0,Y 337.67,Z 723.085,A -85,B 0,C 180,E1 15432.692,E2 15432.692} C_VEL
LIN {X 0,Y 332.108,Z 741.486,A -85,B 0,C 180,E1 15430.336,E2 15430.336} C_VEL
LIN {X 0,Y 326.712,Z 758.318,A -85,B 0,C 180,E1 15427.738,E2 15427.738} C_VEL
LIN {X 0,Y 321.378,Z 774.656,A -85,B 0,C 180,E1 15424.703,E2 15424.703} C_VEL
LIN {X 0,Y 316.778,Z 788.834,A -85,B 0,C 180,E1 15421.548,E2 15421.548} C_VEL
LIN {X 0,Y 312.668,Z 801.916,A -85,B 0,C 180,E1 15418.039,E2 15418.039} C_VEL
LIN {X 0,Y 309.434,Z 813.014,A -85,B 0,C 180,E1 15414.43,E2 15414.43} C_VEL
LIN {X 0,Y 306.874,Z 823.178,A -85,B 0,C 180,E1 15410.403,E2 15410.403} C_VEL
LIN {X 0,Y 305.313,Z 831.004,A -85,B 0,C 180,E1 15406.553,E2 15406.553} C_VEL
LIN {X 0,Y 304.446,Z 837.018,A -85,B 0,C 180,E1 15402.711,E2 15402.711} C_VEL
LIN {X 0,Y 304.093,Z 841.615,A -85,B 0,C 180,E1 15398.699,E2 15398.699} C_VEL
LIN {X 0,Y 304.057,Z 844.207,A -85,B 0,C 180,E1 15395.283,E2 15395.283} C_VEL
LIN {X 0,Y 304.085,Z 845.568,A -85,B 0,C 180,E1 15391.507,E2 15391.507} C_VEL
LIN {X 0,Y 304.083,Z 845.542,A -85,B 0,C 180,E1 15388.304,E2 15388.304} C_VEL
LIN {X 0,Y 304.056,Z 844.077,A -85,B 0,C 180,E1 15384.528,E2 15384.528} C_VEL
LIN {X 0,Y 304.098,Z 841.432,A -85,B 0,C 180,E1 15381.111,E2 15381.111} C_VEL
LIN {X 0,Y 304.475,Z 836.734,A -85,B 0,C 180,E1 15377.097,E2 15377.097} C_VEL
LIN {X 0,Y 305.372,Z 830.659,A -85,B 0,C 180,E1 15373.254,E2 15373.254} C_VEL
LIN {X 0,Y 306.973,Z 822.726,A -85,B 0,C 180,E1 15369.405,E2 15369.405} C_VEL
LIN {X 0,Y 309.432,Z 812.984,A -85,B 0,C 180,E1 15365.569,E2 15365.569} C_VEL
LIN {X 0,Y 312.669,Z 801.865,A -85,B 0,C 180,E1 15361.957,E2 15361.957} C_VEL
LIN {X 0,Y 316.586,Z 789.354,A -85,B 0,C 180,E1 15358.594,E2 15358.594} C_VEL
LIN {X 0,Y 321.078,Z 775.477,A -85,B 0,C 180,E1 15355.477,E2 15355.477} C_VEL
LIN {X 0,Y 326.144,Z 760.029,A -85,B 0,C 180,E1 15352.562,E2 15352.562} C_VEL
LIN {X 0,Y 331.533,Z 743.265,A -85,B 0,C 180,E1 15349.919,E2 15349.919} C_VEL
LIN {X 0,Y 336.825,Z 725.724,A -85,B 0,C 180,E1 15347.637,E2 15347.637} C_VEL
LIN {X 0,Y 342.11,Z 706.982,A -85,B 0,C 180,E1 15345.615,E2 15345.615} C_VEL
LIN {X 0,Y 346.999,Z 687.885,A -85,B 0,C 180,E1 15343.917,E2 15343.917} C_VEL
LIN {X 0,Y 351.63,Z 667.325,A -85,B 0,C 180,E1 15342.45,E2 15342.45} C_VEL
LIN {X 0,Y 355.434,Z 647.085,A -85,B 0,C 180,E1 15341.317,E2 15341.317} C_VEL
LIN {X 0,Y 358.836,Z 624.904,A -85,B 0,C 180,E1 15340.377,E2 15340.377} C_VEL
LIN {X 0,Y 361.239,Z 603.3,A -85,B 0,C 180,E1 15339.717,E2 15339.717} C_VEL
LIN {X 0,Y 372.237,Z 411.837,A -85,B 0,C 180,E1 15335.704,E2 15335.704} C_VEL
LIN {X 0,Y 373.533,Z 386.944,A -85,B 0,C 180,E1 15335.165,E2 15335.165} C_VEL
LIN {X 0,Y 364.479,Z 371.721,A -85,B 0,C 180,E1 15332.759,E2 15332.759} C_VEL
LIN {X 0,Y 355.848,Z 358.298,A -85,B 0,C 180,E1 15330.242,E2 15330.242} C_VEL
LIN {X 0,Y 348.146,Z 347.387,A -85,B 0,C 180,E1 15327.773,E2 15327.773} C_VEL
LIN {X 0,Y 341.691,Z 338.59,A -85,B 0,C 180,E1 15325.477,E2 15325.477} C_VEL
LIN {X 0,Y 334.079,Z 328.942,A -85,B 0,C 180,E1 15322.432,E2 15322.432} C_VEL
LIN {X 0,Y 329.623,Z 323.525,A -85,B 0,C 180,E1 15320.416,E2 15320.416} C_VEL
LIN {X 0,Y 324.903,Z 317.875,A -85,B 0,C 180,E1 15318.015,E2 15318.015} C_VEL
LIN {X 0,Y 321.274,Z 313.893,A -85,B 0,C 180,E1 15315.941,E2 15315.941} C_VEL
LIN {X 0,Y 320.112,Z 312.094,A -85,B 0,C 180,E1 15315.025,E2 15315.025} C_VEL
LIN {X 0,Y 317.667,Z 308.376,A -85,B 0,C 180,E1 15311.989,E2 15311.989} C_VEL
LIN {X 0,Y 316.834,Z 306.656,A -85,B 0,C 180,E1 15310.546,E2 15310.546} C_VEL
LIN {X 0,Y 313.768,Z 301.475,A -85,B 0,C 180,E1 15303.288,E2 15303.288} C_VEL
LIN {X 0,Y 313.001,Z 300.745,A -85,B 0,C 180,E1 15297.986,E2 15297.986} C_VEL
LIN {X 0,Y 313.835,Z 301.572,A -85,B 0,C 180,E1 15293.046,E2 15293.046} C_VEL
LIN {X 0,Y 317.189,Z 307.222,A -85,B 0,C 180,E1 15285.393,E2 15285.393} C_VEL
LIN {X 0,Y 319.165,Z 311.179,A -85,B 0,C 180,E1 15282.309,E2 15282.309} C_VEL
LIN {X 0,Y 320.256,Z 312.72,A -85,B 0,C 180,E1 15281.077,E2 15281.077} C_VEL
LIN {X 0,Y 322.492,Z 316.74,A -85,B 0,C 180,E1 15278.54,E2 15278.54} C_VEL
LIN {X 0,Y 324.294,Z 320.011,A -85,B 0,C 180,E1 15276.996,E2 15276.996} C_VEL
LIN {X 0,Y 327.496,Z 323.88,A -85,B 0,C 180,E1 15275.323,E2 15275.323} C_VEL
LIN {X 0,Y 331.46,Z 328.865,A -85,B 0,C 180,E1 15273.435,E2 15273.435} C_VEL
LIN {X 0,Y 336.383,Z 335.335,A -85,B 0,C 180,E1 15271.312,E2 15271.312} C_VEL
LIN {X 0,Y 342.51,Z 343.745,A -85,B 0,C 180,E1 15268.937,E2 15268.937} C_VEL
LIN {X 0,Y 348.993,Z 352.986,A -85,B 0,C 180,E1 15266.676,E2 15266.676} C_VEL
LIN {X 0,Y 357.91,Z 366.631,A -85,B 0,C 180,E1 15263.882,E2 15263.882} C_VEL
LIN {X 0,Y 367.943,Z 383.572,A -85,B 0,C 180,E1 15261.067,E2 15261.067} C_VEL
LIN {X 0,Y 371.401,Z 390.2,A -85,B 0,C 180,E1 15260.149,E2 15260.149} C_VEL
LIN {X 0,Y 361.085,Z 596.551,A -85,B 0,C 180,E1 15256.12,E2 15256.12} C_VEL
LIN {X 0,Y 358.863,Z 617.722,A -85,B 0,C 180,E1 15255.467,E2 15255.467} C_VEL
LIN {X 0,Y 355.958,Z 637.349,A -85,B 0,C 180,E1 15254.605,E2 15254.605} C_VEL
LIN {X 0,Y 352.09,Z 657.84,A -85,B 0,C 180,E1 15253.41,E2 15253.41} C_VEL
LIN {X 0,Y 347.879,Z 676.264,A -85,B 0,C 180,E1 15252.041,E2 15252.041} C_VEL
LIN {X 0,Y 342.974,Z 694.701,A -85,B 0,C 180,E1 15250.329,E2 15250.329} C_VEL
LIN {X 0,Y 337.919,Z 711.372,A -85,B 0,C 180,E1 15248.414,E2 15248.414} C_VEL
LIN {X 0,Y 332.657,Z 727.302,A -85,B 0,C 180,E1 15246.196,E2 15246.196} C_VEL
LIN {X 0,Y 327.518,Z 741.847,A -85,B 0,C 180,E1 15243.752,E2 15243.752} C_VEL
LIN {X 0,Y 322.474,Z 755.503,A -85,B 0,C 180,E1 15240.976,E2 15240.976} C_VEL
LIN {X 0,Y 317.632,Z 768.222,A -85,B 0,C 180,E1 15237.804,E2 15237.804} C_VEL
LIN {X 0,Y 313.538,Z 779.043,A -85,B 0,C 180,E1 15234.491,E2 15234.491} C_VEL
LIN {X 0,Y 310.025,Z 788.822,A -85,B 0,C 180,E1 15230.778,E2 15230.778} C_VEL
LIN {X 0,Y 307.475,Z 796.643,A -85,B 0,C 180,E1 15227.017,E2 15227.017} C_VEL
LIN {X 0,Y 305.777,Z 802.719,A -85,B 0,C 180,E1 15223.232,E2 15223.232} C_VEL
LIN {X 0,Y 304.774,Z 807.276,A -85,B 0,C 180,E1 15219.25,E2 15219.25} C_VEL
LIN {X 0,Y 304.315,Z 810.082,A -85,B 0,C 180,E1 15215.41,E2 15215.41} C_VEL
LIN {X 0,Y 304.168,Z 811.451,A -85,B 0,C 180,E1 15211.507,E2 15211.507} C_VEL
LIN {X 0,Y 304.18,Z 811.379,A -85,B 0,C 180,E1 15207.739,E2 15207.739} C_VEL
LIN {X 0,Y 304.352,Z 809.795,A -85,B 0,C 180,E1 15203.966,E2 15203.966} C_VEL
LIN {X 0,Y 304.897,Z 806.612,A -85,B 0,C 180,E1 15199.991,E2 15199.991} C_VEL
LIN {X 0,Y 306.019,Z 801.781,A -85,B 0,C 180,E1 15196.024,E2 15196.024} C_VEL
LIN {X 0,Y 307.867,Z 795.478,A -85,B 0,C 180,E1 15192.225,E2 15192.225} C_VEL
LIN {X 0,Y 310.584,Z 787.311,A -85,B 0,C 180,E1 15188.47,E2 15188.47} C_VEL
LIN {X 0,Y 314.065,Z 777.688,A -85,B 0,C 180,E1 15184.95,E2 15184.95} C_VEL
LIN {X 0,Y 318.408,Z 766.204,A -85,B 0,C 180,E1 15181.553,E2 15181.553} C_VEL
LIN {X 0,Y 318.66,Z 765.546,A -85,B 0,C 180,E1 15181.378,E2 15181.378} C_VEL
LIN {X 0,Y 319.412,Z 761.41,A -85,B 0,C 180,E1 15180.205,E2 15180.205} C_VEL
LIN {X 0,Y 318.473,Z 750.833,A -85,B 0,C 180,E1 15177.133,E2 15177.133} C_VEL
LIN {X 0,Y 319.478,Z 746.033,A -85,B 0,C 180,E1 15176.053,E2 15176.053} C_VEL
LIN {X 0,Y 325.004,Z 731.37,A -85,B 0,C 180,E1 15173.414,E2 15173.414} C_VEL
LIN {X 0,Y 330.692,Z 715.182,A -85,B 0,C 180,E1 15171.033,E2 15171.033} C_VEL
LIN {X 0,Y 336.073,Z 698.249,A -85,B 0,C 180,E1 15169.005,E2 15169.005} C_VEL
LIN {X 0,Y 341.145,Z 680.364,A -85,B 0,C 180,E1 15167.257,E2 15167.257} C_VEL
LIN {X 0,Y 345.69,Z 662.008,A -85,B 0,C 180,E1 15165.81,E2 15165.81} C_VEL
LIN {X 0,Y 349.689,Z 642.728,A -85,B 0,C 180,E1 15164.607,E2 15164.607} C_VEL
LIN {X 0,Y 352.952,Z 622.544,A -85,B 0,C 180,E1 15163.658,E2 15163.658} C_VEL
LIN {X 0,Y 355.378,Z 601.874,A -85,B 0,C 180,E1 15162.959,E2 15162.959} C_VEL
LIN {X 0,Y 357.182,Z 574.388,A -85,B 0,C 180,E1 15162.351,E2 15162.351} C_VEL
LIN {X 0,Y 366.427,Z 393.393,A -85,B 0,C 180,E1 15158.798,E2 15158.798} C_VEL
LIN {X 0,Y 357.13,Z 377.062,A -85,B 0,C 180,E1 15156.16,E2 15156.16} C_VEL
LIN {X 0,Y 348.239,Z 362.86,A -85,B 0,C 180,E1 15153.356,E2 15153.356} C_VEL
LIN {X 0,Y 341.146,Z 352.391,A -85,B 0,C 180,E1 15150.858,E2 15150.858} C_VEL
LIN {X 0,Y 335.367,Z 344.144,A -85,B 0,C 180,E1 15148.589,E2 15148.589} C_VEL
LIN {X 0,Y 331.264,Z 338.703,A -85,B 0,C 180,E1 15146.824,E2 15146.824} C_VEL
LIN {X 0,Y 327.44,Z 333.612,A -85,B 0,C 180,E1 15145.019,E2 15145.019} C_VEL
LIN {X 0,Y 323.731,Z 328.95,A -85,B 0,C 180,E1 15143.095,E2 15143.095} C_VEL
LIN {X 0,Y 320.086,Z 324.176,A -85,B 0,C 180,E1 15140.957,E2 15140.957} C_VEL
LIN {X 0,Y 316.568,Z 319.902,A -85,B 0,C 180,E1 15138.603,E2 15138.603} C_VEL
LIN {X 0,Y 315.219,Z 318.193,A -85,B 0,C 180,E1 15137.538,E2 15137.538} C_VEL
LIN {X 0,Y 313.108,Z 314.544,A -85,B 0,C 180,E1 15134.612,E2 15134.612} C_VEL
LIN {X 0,Y 312.257,Z 313.083,A -85,B 0,C 180,E1 15133.141,E2 15133.141} C_VEL
LIN {X 0,Y 309.717,Z 308.408,A -85,B 0,C 180,E1 15126.116,E2 15126.116} C_VEL
LIN {X 0,Y 309.159,Z 307.831,A -85,B 0,C 180,E1 15120.927,E2 15120.927} C_VEL
LIN {X 0,Y 309.861,Z 308.656,A -85,B 0,C 180,E1 15116.671,E2 15116.671} C_VEL
LIN {X 0,Y 313.242,Z 313.904,A -85,B 0,C 180,E1 15109.331,E2 15109.331} C_VEL
LIN {X 0,Y 317.06,Z 318.727,A -85,B 0,C 180,E1 15106.236,E2 15106.236} C_VEL
LIN {X 0,Y 319.104,Z 320.639,A -85,B 0,C 180,E1 15104.88,E2 15104.88} C_VEL
LIN {X 0,Y 322.677,Z 325.047,A -85,B 0,C 180,E1 15102.695,E2 15102.695} C_VEL
LIN {X 0,Y 324.365,Z 326.895,A -85,B 0,C 180,E1 15101.768,E2 15101.768} C_VEL
LIN {X 0,Y 329.365,Z 333.017,A -85,B 0,C 180,E1 15099.242,E2 15099.242} C_VEL
LIN {X 0,Y 336.421,Z 341.89,A -85,B 0,C 180,E1 15096.159,E2 15096.159} C_VEL
LIN {X 0,Y 344.314,Z 352.665,A -85,B 0,C 180,E1 15093.157,E2 15093.157} C_VEL
LIN {X 0,Y 351.897,Z 363.582,A -85,B 0,C 180,E1 15090.604,E2 15090.604} C_VEL
LIN {X 0,Y 360.504,Z 377.05,A -85,B 0,C 180,E1 15087.989,E2 15087.989} C_VEL
LIN {X 0,Y 368.667,Z 391.015,A -85,B 0,C 180,E1 15085.718,E2 15085.718} C_VEL
LIN {X 0,Y 356.307,Z 599.02,A -85,B 0,C 180,E1 15081.353,E2 15081.353} C_VEL
LIN {X 0,Y 353.85,Z 622.345,A -85,B 0,C 180,E1 15080.677,E2 15080.677} C_VEL
LIN {X 0,Y 350.672,Z 643.337,A -85,B 0,C 180,E1 15079.829,E2 15079.829} C_VEL
LIN {X 0,Y 346.957,Z 662.87,A -85,B 0,C 180,E1 15078.775,E2 15078.775} C_VEL
LIN {X 0,Y 342.371,Z 683.197,A -85,B 0,C 180,E1 15077.385,E2 15077.385} C_VEL
LIN {X 0,Y 337.328,Z 702.73,A -85,B 0,C 180,E1 15075.726,E2 15075.726} C_VEL
LIN {X 0,Y 331.859,Z 721.709,A -85,B 0,C 180,E1 15073.744,E2 15073.744} C_VEL
LIN {X 0,Y 326.428,Z 739.012,A -85,B 0,C 180,E1 15071.539,E2 15071.539} C_VEL
LIN {X 0,Y 320.537,Z 756.711,A -85,B 0,C 180,E1 15068.827,E2 15068.827} C_VEL
LIN {X 0,Y 315.19,Z 772.368,A -85,B 0,C 180,E1 15065.934,E2 15065.934} C_VEL
LIN {X 0,Y 310.225,Z 786.787,A -85,B 0,C 180,E1 15062.733,E2 15062.733} C_VEL
LIN {X 0,Y 305.967,Z 799.417,A -85,B 0,C 180,E1 15059.351,E2 15059.351} C_VEL
LIN {X 0,Y 302.204,Z 811.438,A -85,B 0,C 180,E1 15055.474,E2 15055.474} C_VEL
LIN {X 0,Y 299.589,Z 820.981,A -85,B 0,C 180,E1 15051.743,E2 15051.743} C_VEL
LIN {X 0,Y 297.716,Z 829.081,A -85,B 0,C 180,E1 15047.795,E2 15047.795} C_VEL
LIN {X 0,Y 296.594,Z 835.737,A -85,B 0,C 180,E1 15043.649,E2 15043.649} C_VEL
LIN {X 0,Y 296.146,Z 840.468,A -85,B 0,C 180,E1 15039.718,E2 15039.718} C_VEL
LIN {X 0,Y 296.057,Z 843.388,A -85,B 0,C 180,E1 15036.009,E2 15036.009} C_VEL
LIN {X 0,Y 296.089,Z 845.018,A -85,B 0,C 180,E1 15032.322,E2 15032.322} C_VEL
LIN {X 0,Y 296.104,Z 845.168,A -85,B 0,C 180,E1 15028.839,E2 15028.839} C_VEL
LIN {X 0,Y 296.066,Z 844.091,A -85,B 0,C 180,E1 15025.157,E2 15025.157} C_VEL
LIN {X 0,Y 296.094,Z 841.492,A -85,B 0,C 180,E1 15021.456,E2 15021.456} C_VEL
LIN {X 0,Y 296.411,Z 837.354,A -85,B 0,C 180,E1 15017.533,E2 15017.533} C_VEL
LIN {X 0,Y 297.257,Z 831.489,A -85,B 0,C 180,E1 15013.588,E2 15013.588} C_VEL
LIN {X 0,Y 298.927,Z 823.53,A -85,B 0,C 180,E1 15009.439,E2 15009.439} C_VEL
LIN {X 0,Y 301.284,Z 814.654,A -85,B 0,C 180,E1 15005.701,E2 15005.701} C_VEL
LIN {X 0,Y 304.728,Z 803.261,A -85,B 0,C 180,E1 15001.805,E2 15001.805} C_VEL
LIN {X 0,Y 308.74,Z 791.028,A -85,B 0,C 180,E1 14998.357,E2 14998.357} C_VEL
LIN {X 0,Y 313.647,Z 776.692,A -85,B 0,C 180,E1 14994.985,E2 14994.985} C_VEL
LIN {X 0,Y 318.962,Z 761.345,A -85,B 0,C 180,E1 14991.979,E2 14991.979} C_VEL
LIN {X 0,Y 324.642,Z 744.412,A -85,B 0,C 180,E1 14989.238,E2 14989.238} C_VEL
LIN {X 0,Y 330.123,Z 727.15,A -85,B 0,C 180,E1 14986.924,E2 14986.924} C_VEL
LIN {X 0,Y 335.662,Z 708.505,A -85,B 0,C 180,E1 14984.852,E2 14984.852} C_VEL
LIN {X 0,Y 340.875,Z 689.138,A -85,B 0,C 180,E1 14983.084,E2 14983.084} C_VEL
LIN {X 0,Y 345.595,Z 668.972,A -85,B 0,C 180,E1 14981.618,E2 14981.618} C_VEL
LIN {X 0,Y 349.702,Z 648.276,A -85,B 0,C 180,E1 14980.427,E2 14980.427} C_VEL
LIN {X 0,Y 353.203,Z 626.682,A -85,B 0,C 180,E1 14979.485,E2 14979.485} C_VEL
LIN {X 0,Y 355.82,Z 604.614,A -85,B 0,C 180,E1 14978.791,E2 14978.791} C_VEL
LIN {X 0,Y 361.101,Z 516.806,A -85,B 0,C 180,E1 14976.907,E2 14976.907} C_VEL
LIN {X 0,Y 368.498,Z 390.727,A -85,B 0,C 180,E1 14974.264,E2 14974.264} C_VEL
LIN {X 0,Y 359.511,Z 375.483,A -85,B 0,C 180,E1 14971.758,E2 14971.758} C_VEL
LIN {X 0,Y 351.118,Z 362.474,A -85,B 0,C 180,E1 14969.186,E2 14969.186} C_VEL
LIN {X 0,Y 343.055,Z 350.857,A -85,B 0,C 180,E1 14966.436,E2 14966.436} C_VEL
LIN {X 0,Y 335.417,Z 340.724,A -85,B 0,C 180,E1 14963.497,E2 14963.497} C_VEL
LIN {X 0,Y 330.878,Z 335.06,A -85,B 0,C 180,E1 14961.54,E2 14961.54} C_VEL
LIN {X 0,Y 327.599,Z 330.885,A -85,B 0,C 180,E1 14959.988,E2 14959.988} C_VEL
LIN {X 0,Y 323.136,Z 325.426,A -85,B 0,C 180,E1 14957.652,E2 14957.652} C_VEL
LIN {X 0,Y 319.453,Z 321.234,A -85,B 0,C 180,E1 14955.475,E2 14955.475} C_VEL
LIN {X 0,Y 318.205,Z 319.633,A -85,B 0,C 180,E1 14954.652,E2 14954.652} C_VEL
LIN {X 0,Y 314.43,Z 315.794,A -85,B 0,C 180,E1 14951.928,E2 14951.928} C_VEL
LIN {X 0,Y 312.831,Z 313.578,A -85,B 0,C 180,E1 14950.496,E2 14950.496} C_VEL
LIN {X 0,Y 309.7,Z 308.338,A -85,B 0,C 180,E1 14943.146,E2 14943.146} C_VEL
LIN {X 0,Y 308.963,Z 307.652,A -85,B 0,C 180,E1 14937.96,E2 14937.96} C_VEL
LIN {X 0,Y 309.806,Z 308.512,A -85,B 0,C 180,E1 14932.955,E2 14932.955} C_VEL
LIN {X 0,Y 312.948,Z 314.055,A -85,B 0,C 180,E1 14925.477,E2 14925.477} C_VEL
LIN {X 0,Y 315.025,Z 318.029,A -85,B 0,C 180,E1 14922.355,E2 14922.355} C_VEL
LIN {X 0,Y 316.4,Z 319.673,A -85,B 0,C 180,E1 14921.291,E2 14921.291} C_VEL
LIN {X 0,Y 319.777,Z 323.912,A -85,B 0,C 180,E1 14919.022,E2 14919.022} C_VEL
LIN {X 0,Y 321.815,Z 326.495,A -85,B 0,C 180,E1 14917.795,E2 14917.795} C_VEL
LIN {X 0,Y 325.883,Z 331.725,A -85,B 0,C 180,E1 14915.579,E2 14915.579} C_VEL
LIN {X 0,Y 329.357,Z 336.162,A -85,B 0,C 180,E1 14913.884,E2 14913.884} C_VEL
LIN {X 0,Y 334.282,Z 342.766,A -85,B 0,C 180,E1 14911.7,E2 14911.7} C_VEL
LIN {X 0,Y 340.104,Z 350.959,A -85,B 0,C 180,E1 14909.38,E2 14909.38} C_VEL
LIN {X 0,Y 346.373,Z 360.058,A -85,B 0,C 180,E1 14907.133,E2 14907.133} C_VEL
LIN {X 0,Y 354.856,Z 373.383,A -85,B 0,C 180,E1 14904.394,E2 14904.394} C_VEL
LIN {X 0,Y 364.225,Z 389.484,A -85,B 0,C 180,E1 14901.679,E2 14901.679} C_VEL
LIN {X 0,Y 366.402,Z 393.712,A -85,B 0,C 180,E1 14901.077,E2 14901.077} C_VEL
LIN {X 0,Y 355.811,Z 596.594,A -85,B 0,C 180,E1 14897.084,E2 14897.084} C_VEL
LIN {X 0,Y 353.518,Z 617.738,A -85,B 0,C 180,E1 14896.43,E2 14896.43} C_VEL
LIN {X 0,Y 350.477,Z 637.625,A -85,B 0,C 180,E1 14895.554,E2 14895.554} C_VEL
LIN {X 0,Y 346.522,Z 657.878,A -85,B 0,C 180,E1 14894.367,E2 14894.367} C_VEL
LIN {X 0,Y 342.237,Z 676.076,A -85,B 0,C 180,E1 14893.013,E2 14893.013} C_VEL
LIN {X 0,Y 337.135,Z 694.561,A -85,B 0,C 180,E1 14891.289,E2 14891.289} C_VEL
LIN {X 0,Y 331.877,Z 711.314,A -85,B 0,C 180,E1 14889.358,E2 14889.358} C_VEL
LIN {X 0,Y 326.4,Z 727.298,A -85,B 0,C 180,E1 14887.118,E2 14887.118} C_VEL
LIN {X 0,Y 321.197,Z 741.47,A -85,B 0,C 180,E1 14884.726,E2 14884.726} C_VEL
LIN {X 0,Y 315.874,Z 755.199,A -85,B 0,C 180,E1 14881.911,E2 14881.911} C_VEL
LIN {X 0,Y 310.961,Z 767.489,A -85,B 0,C 180,E1 14878.835,E2 14878.835} C_VEL
LIN {X 0,Y 306.606,Z 778.424,A -85,B 0,C 180,E1 14875.496,E2 14875.496} C_VEL
LIN {X 0,Y 302.954,Z 787.98,A -85,B 0,C 180,E1 14871.896,E2 14871.896} C_VEL
LIN {X 0,Y 300.092,Z 796.102,A -85,B 0,C 180,E1 14868.05,E2 14868.05} C_VEL
LIN {X 0,Y 298.069,Z 802.635,A -85,B 0,C 180,E1 14863.976,E2 14863.976} C_VEL
LIN {X 0,Y 296.948,Z 807.15,A -85,B 0,C 180,E1 14860.084,E2 14860.084} C_VEL
LIN {X 0,Y 296.373,Z 810.289,A -85,B 0,C 180,E1 14856.003,E2 14856.003} C_VEL
LIN {X 0,Y 296.197,Z 811.837,A -85,B 0,C 180,E1 14852.128,E2 14852.128} C_VEL
LIN {X 0,Y 296.177,Z 811.911,A -85,B 0,C 180,E1 14848.452,E2 14848.452} C_VEL
LIN {X 0,Y 296.337,Z 810.561,A -85,B 0,C 180,E1 14844.385,E2 14844.385} C_VEL
LIN {X 0,Y 296.825,Z 807.84,A -85,B 0,C 180,E1 14840.5,E2 14840.5} C_VEL
LIN {X 0,Y 297.895,Z 803.305,A -85,B 0,C 180,E1 14836.412,E2 14836.412} C_VEL
